    |   movel(p[0.465893, -0.053931, -0.000100, 0.000000, -3.141593, 0.000000],accel_mss,speed_ms,0,0.000)
    |   movel(p[0.464835, -0.052791, -0.000100, 0.000000, -3.141593, 0.000000],accel_mss,speed_ms,0,0.001)
    |   movel(p[0.463851, -0.051647, -0.000100, 0.000000, -3.141593, 0.000000],accel_mss,speed_ms,0,0.001)
    |   movel(p[0.463361, -0.050896, -0.000100, 0.000000, -3.141593, 0.000000],accel_mss,speed_ms,0,0.000)
    |   movel(p[0.463213, -0.050560, -0.000100, 0.000000, -3.141593, 0.000000],accel_mss,speed_ms,0,0.000)
    |   movel(p[0.463098, -0.050199, -0.000100, 0.000000, -3.141593, 0.000000],accel_mss,speed_ms,0,0.000)
    |   movel(p[0.463025, -0.049844, -0.000100, 0.000000, -3.141593, 0.000000],accel_mss,speed_ms,0,0.000)
    |   movel(p[0.463001, -0.049520, -0.000100, 0.000000, -3.141593, 0.000000],accel_mss,speed_ms,0,0.000)
    |   movel(p[0.462988, -0.049209, -0.000100, 0.000000, -3.141593, 0.000000],accel_mss,speed_ms,0,0.000)
    |   movel(p[0.462948, -0.048819, -0.000100, 0.000000, -3.141593, 0.000000],accel_mss,speed_ms,0,0.000)
    |   movel(p[0.462890, -0.048420, -0.000100, 0.000000, 3.141593, 0.000000],accel_mss,speed_ms,0,0.000)
    |   movel(p[0.462821, -0.048073, -0.000100, 0.000000, 3.141593, 0.000000],accel_mss,speed_ms,0,0.000)
    |   movel(p[0.462724, -0.047613, -0.000100, 0.000000, -3.141593, 0.000000],accel_mss,speed_ms,0,0.000)
    |   movel(p[0.462714, -0.047386, -0.000100, 0.000000, 3.141593, 0.000000],accel_mss,speed_ms,0,0.000)
    |   movel(p[0.462774, -0.047234, -0.000100, 0.000000, -3.141593, 0.000000],accel_mss,speed_ms,0,0.000)
    |   movel(p[0.462918, -0.047091, -0.000100, 0.000000, -3.141593, 0.000000],accel_mss,speed_ms,0,0.000)
    |   movel(p[0.463032, -0.047019, -0.000100, 0.000000, -3.141593, 0.000000],accel_mss,speed_ms,0,0.000)
    |   movel(p[0.463146, -0.046968, -0.000100, 0.000000, -3.141593, 0.000000],accel_mss,speed_ms,0,0.000)
    |   movel(p[0.463245, -0.046945, -0.000100, 0.000000, -3.141593, 0.000000],accel_mss,speed_ms,0,0.000)
    |   movel(p[0.463376, -0.046956, -0.000100, 0.000000, -3.141593, 0.000000],accel_mss,speed_ms,0,0.000)
    |   movel(p[0.463547, -0.046827, -0.000100, 0.000000, -3.141593, 0.000000],accel_mss,speed_ms,0,0.000)
    |   movel(p[0.463749, -0.046646, -0.000100, 0.000000, -3.141593, 0.000000],accel_mss,speed_ms,0,0.000)
    |   movel(p[0.463969, -0.046417, -0.000100, 0.000000, -3.141593, 0.000000],accel_mss,speed_ms,0,0.000)
    |   movel(p[0.464381, -0.046019, -0.000100, 0.000000, -3.141593, 0.000000],accel_mss,speed_ms,0,0.000)
    |   movel(p[0.464651, -0.045948, -0.000100, 0.000000, 3.141593, 0.000000],accel_mss,speed_ms,0,0.000)
    |   movel(p[0.464889, -0.046112, -0.000100, 0.000000, -3.141593, 0.000000],accel_mss,speed_ms,0,0.000)
    |   movel(p[0.465184, -0.046650, -0.000100, 0.000000, -3.141593, 0.000000],accel_mss,speed_ms,0,0.000)
    |   movel(p[0.465308, -0.047062, -0.000100, 0.000000, 3.141593, 0.000000],accel_mss,speed_ms,0,0.000)
    |   movel(p[0.465283, -0.047444, -0.000100, 0.000000, 3.141593, 0.000000],accel_mss,speed_ms,0,0.000)
    |   movel(p[0.465098, -0.047820, -0.000100, 0.000000, -3.141593, 0.000000],accel_mss,speed_ms,0,0.000)
    |   movel(p[0.464742, -0.048218, -0.000100, 0.000000, -3.141593, 0.000000],accel_mss,speed_ms,0,0.000)
    |   movel(p[0.464491, -0.048534, -0.000100, 0.000000, -3.141593, 0.000000],accel_mss,speed_ms,0,0.000)
    |   movel(p[0.464362, -0.048895, -0.000100, 0.000000, -3.141593, 0.000000],accel_mss,speed_ms,0,0.000)
    |   movel(p[0.464394, -0.049167, -0.000100, 0.000000, -3.141593, 0.000000],accel_mss,speed_ms,0,0.000)
    |   movel(p[0.464563, -0.049279, -0.000100, 0.000000, -3.141593, 0.000000],accel_mss,speed_ms,0,0.000)
    |   movel(p[0.464679, -0.049242, -0.000100, 0.000000, -3.141593, 0.000000],accel_mss,speed_ms,0,0.000)
    |   movel(p[0.464892, -0.049075, -0.000100, 0.000000, 3.141593, 0.000000],accel_mss,speed_ms,0,0.000)
    |   movel(p[0.465136, -0.048852, -0.000100, 0.000000, -3.141593, 0.000000],accel_mss,speed_ms,0,0.000)
    |   movel(p[0.465385, -0.048586, -0.000100, 0.000000, 3.141593, 0.000000],accel_mss,speed_ms,0,0.000)
    |   movel(p[0.465794, -0.048130, -0.000100, 0.000000, -3.141593, 0.000000],accel_mss,speed_ms,0,0.000)
    |   movel(p[0.465936, -0.048028, -0.000100, 0.000000, 3.141593, 0.000000],accel_mss,speed_ms,0,0.000)
    |   movel(p[0.466037, -0.048055, -0.000100, 0.000000, -3.141593, 0.000000],accel_mss,speed_ms,0,0.000)
    |   movel(p[0.466147, -0.048249, -0.000100, 0.000000, 3.141593, 0.000000],accel_mss,speed_ms,0,0.000)
    |   movel(p[0.466218, -0.048402, -0.000100, 0.000000, -3.141593, 0.000000],accel_mss,speed_ms,0,0.000)
    |   movel(p[0.466305, -0.048569, -0.000100, 0.000000, -3.141593, 0.000000],accel_mss,speed_ms,0,0.000)
    |   movel(p[0.466394, -0.048724, -0.000100, 0.000000, -3.141593, 0.000000],accel_mss,speed_ms,0,0.000)
    |   movel(p[0.466470, -0.048840, -0.000100, 0.000000, -3.141593, 0.000000],accel_mss,speed_ms,0,0.000)
    |   movel(p[0.466537, -0.048985, -0.000100, 0.000000, -3.141593, 0.000000],accel_mss,speed_ms,0,0.000)
    |   movel(p[0.466547, -0.049150, -0.000100, 0.000000, -3.141593, 0.000000],accel_mss,speed_ms,0,0.000)
    |   movel(p[0.466496, -0.049362, -0.000100, 0.000000, -3.141593, 0.000000],accel_mss,speed_ms,0,0.000)
    |   movel(p[0.466370, -0.049665, -0.000100, 0.000000, -3.141593, 0.000000],accel_mss,speed_ms,0,0.000)
    |   movel(p[0.466251, -0.049909, -0.000100, 0.000000, 3.141593, 0.000000],accel_mss,speed_ms,0,0.000)
    |   movel(p[0.466117, -0.050154, -0.000100, 0.000000, -3.141593, 0.000000],accel_mss,speed_ms,0,0.000)
    |   movel(p[0.465988, -0.050369, -0.000100, 0.000000, -3.141593, 0.000000],accel_mss,speed_ms,0,0.000)
    |   movel(p[0.465888, -0.050504, -0.000100, 0.000000, -3.141593, 0.000000],accel_mss,speed_ms,0,0.000)
    |   movel(p[0.465811, -0.050625, -0.000100, 0.000000, -3.141593, 0.000000],accel_mss,speed_ms,0,0.000)
    |   movel(p[0.465753, -0.050783, -0.000100, 0.000000, -3.141593, 0.000000],accel_mss,speed_ms,0,0.000)
    |   movel(p[0.465723, -0.050952, -0.000100, 0.000000, -3.141593, 0.000000],accel_mss,speed_ms,0,0.000)
    |   movel(p[0.465726, -0.051104, -0.000100, 0.000000, -3.141593, 0.000000],accel_mss,speed_ms,0,0.000)
    |   movel(p[0.465772, -0.051280, -0.000100, 0.000000, -3.141593, 0.000000],accel_mss,speed_ms,0,0.000)
    |   movel(p[0.465851, -0.051379, -0.000100, 0.000000, -3.141593, 0.000000],accel_mss,speed_ms,0,0.000)
    |   movel(p[0.465984, -0.051424, -0.000100, 0.000000, -3.141593, 0.000000],accel_mss,speed_ms,0,0.000)
    |   movel(p[0.466209, -0.051423, -0.000100, 0.000000, -3.141593, 0.000000],accel_mss,speed_ms,0,0.000)
    |   movel(p[0.466401, -0.051387, -0.000100, 0.000000, -3.141593, 0.000000],accel_mss,speed_ms,0,0.000)
    |   movel(p[0.466618, -0.051304, -0.000100, 0.000000, 3.141593, 0.000000],accel_mss,speed_ms,0,0.000)
    |   movel(p[0.466827, -0.051191, -0.000100, 0.000000, 3.141593, 0.000000],accel_mss,speed_ms,0,0.000)
    |   movel(p[0.466992, -0.051063, -0.000100, 0.000000, -3.141593, 0.000000],accel_mss,speed_ms,0,0.000)
    |   movel(p[0.467187, -0.050897, -0.000100, 0.000000, 3.141593, 0.000000],accel_mss,speed_ms,0,0.000)
    |   movel(p[0.467319, -0.050833, -0.000100, 0.000000, -3.141593, 0.000000],accel_mss,speed_ms,0,0.000)
    |   movel(p[0.467437, -0.050843, -0.000100, 0.000000, -3.141593, 0.000000],accel_mss,speed_ms,0,0.000)
    |   movel(p[0.467571, -0.050925, -0.000100, 0.000000, -3.141593, 0.000000],accel_mss,speed_ms,0,0.000)
    |   movel(p[0.467659, -0.051011, -0.000100, 0.000000, -3.141593, 0.000000],accel_mss,speed_ms,0,0.000)
    |   movel(p[0.467733, -0.051113, -0.000100, 0.000000, -3.141593, 0.000000],accel_mss,speed_ms,0,0.000)
    |   movel(p[0.467784, -0.051213, -0.000100, 0.000000, 3.141593, 0.000000],accel_mss,speed_ms,0,0.000)
    |   movel(p[0.468014, -0.051722, -0.000100, 0.000000, -3.141593, 0.000000],accel_mss,speed_ms,0,0.000)
    |   movel(p[0.468764, -0.052182, -0.000100, 0.000000, -3.141593, 0.000000],accel_mss,speed_ms,0,0.000)
    |   movel(p[0.469662, -0.052521, -0.000100, 0.000000, 3.141593, 0.000000],accel_mss,speed_ms,0,0.000)
    |   movel(p[0.470426, -0.052584, -0.000100, 0.000000, -3.141593, 0.000000],accel_mss,speed_ms,0,0.000)
    |   movel(p[0.470557, -0.052560, -0.000100, 0.000000, 3.141593, 0.000000],accel_mss,speed_ms,0,0.000)
    |   movel(p[0.470502, -0.052461, -0.000100, 0.000000, -3.141593, 0.000000],accel_mss,speed_ms,0,0.000)
    |   movel(p[0.470257, -0.052349, -0.000100, 0.000000, 3.141593, 0.000000],accel_mss,speed_ms,0,0.000)
    |   movel(p[0.470044, -0.052237, -0.000100, 0.000000, -3.141593, 0.000000],accel_mss,speed_ms,0,0.000)
    |   movel(p[0.469789, -0.052067, -0.000100, 0.000000, -3.141593, 0.000000],accel_mss,speed_ms,0,0.000)
    |   movel(p[0.469535, -0.051871, -0.000100, 0.000000, -3.141593, 0.000000],accel_mss,speed_ms,0,0.000)
    |   movel(p[0.469322, -0.051678, -0.000100, 0.000000, -3.141593, 0.000000],accel_mss,speed_ms,0,0.000)
    |   movel(p[0.469017, -0.051335, -0.000100, 0.000000, -3.141593, 0.000000],accel_mss,speed_ms,0,0.000)
    |   movel(p[0.468787, -0.050993, -0.000100, 0.000000, -3.141593, 0.000000],accel_mss,speed_ms,0,0.000)
    |   movel(p[0.468535, -0.050495, -0.000100, 0.000000, -3.141593, 0.000000],accel_mss,speed_ms,0,0.000)
    |   movel(p[0.468097, -0.049504, -0.000100, 0.000000, -3.141593, 0.000000],accel_mss,speed_ms,0,0.000)
    |   movel(p[0.467644, -0.048482, -0.000100, 0.000000, -3.141593, 0.000000],accel_mss,speed_ms,0,0.000)
    |   movel(p[0.467263, -0.047682, -0.000100, 0.000000, -3.141593, 0.000000],accel_mss,speed_ms,0,0.000)
    |   movel(p[0.466940, -0.047069, -0.000100, 0.000000, -3.141593, 0.000000],accel_mss,speed_ms,0,0.000)
    |   movel(p[0.466677, -0.046654, -0.000100, 0.000000, -3.141593, 0.000000],accel_mss,speed_ms,0,0.000)
    |   movel(p[0.466546, -0.046465, -0.000100, 0.000000, -3.141593, 0.000000],accel_mss,speed_ms,0,0.000)
    |   movel(p[0.466418, -0.046270, -0.000100, 0.000000, -3.141593, 0.000000],accel_mss,speed_ms,0,0.000)
    |   movel(p[0.466311, -0.046095, -0.000100, 0.000000, -3.141593, 0.000000],accel_mss,speed_ms,0,0.000)
    |   movel(p[0.466250, -0.045979, -0.000100, 0.000000, 3.141593, 0.000000],accel_mss,speed_ms,0,0.000)
    |   movel(p[0.466191, -0.045863, -0.000100, 0.000000, -3.141593, 0.000000],accel_mss,speed_ms,0,0.000)
    |   movel(p[0.466091, -0.045688, -0.000100, 0.000000, -3.141593, 0.000000],accel_mss,speed_ms,0,0.000)
    |   movel(p[0.465972, -0.045493, -0.000100, 0.000000, -3.141593, 0.000000],accel_mss,speed_ms,0,0.000)
    |   movel(p[0.465851, -0.045304, -0.000100, 0.000000, -3.141593, 0.000000],accel_mss,speed_ms,0,0.000)
    |   movel(p[0.465728, -0.045110, -0.000100, 0.000000, -3.141593, 0.000000],accel_mss,speed_ms,0,0.000)
    |   movel(p[0.465602, -0.044898, -0.000100, 0.000000, 3.141593, 0.000000],accel_mss,speed_ms,0,0.000)
    |   movel(p[0.465492, -0.044700, -0.000100, 0.000000, -3.141593, 0.000000],accel_mss,speed_ms,0,0.000)
    |   movel(p[0.465420, -0.044554, -0.000100, 0.000000, -3.141593, 0.000000],accel_mss,speed_ms,0,0.000)
    |   movel(p[0.465263, -0.044299, -0.000100, 0.000000, -3.141593, 0.000000],accel_mss,speed_ms,0,0.000)
    |   movel(p[0.465028, -0.044054, -0.000100, 0.000000, -3.141593, 0.000000],accel_mss,speed_ms,0,0.000)
    |   movel(p[0.464698, -0.043807, -0.000100, 0.000000, -3.141593, 0.000000],accel_mss,speed_ms,0,0.000)
    |   movel(p[0.464252, -0.043540, -0.000100, 0.000000, -3.141593, 0.000000],accel_mss,speed_ms,0,0.000)
    |   movel(p[0.463697, -0.043350, -0.000100, 0.000000, -3.141593, 0.000000],accel_mss,speed_ms,0,0.000)
    |   movel(p[0.462896, -0.043284, -0.000100, 0.000000, -3.141593, 0.000000],accel_mss,speed_ms,0,0.000)
    |   movel(p[0.461992, -0.043334, -0.000100, 0.000000, -3.141593, 0.000000],accel_mss,speed_ms,0,0.000)
    |   movel(p[0.461101, -0.043504, -0.000100, 0.000000, -3.141593, 0.000000],accel_mss,speed_ms,0,0.000)
    |   movel(p[0.460265, -0.043707, -0.000100, 0.000000, -3.141593, 0.000000],accel_mss,speed_ms,0,0.000)
    |   movel(p[0.460020, -0.043670, -0.000100, 0.000000, 3.141593, 0.000000],accel_mss,speed_ms,0,0.000)
    |   movel(p[0.459904, -0.043483, -0.000100, 0.000000, -3.141593, 0.000000],accel_mss,speed_ms,0,0.000)
    |   movel(p[0.459894, -0.042823, -0.000100, 0.000000, -3.141593, 0.000000],accel_mss,speed_ms,0,0.000)
    |   movel(p[0.459902, -0.042370, -0.000100, 0.000000, -3.141593, 0.000000],accel_mss,speed_ms,0,0.000)
    |   movel(p[0.459911, -0.041917, -0.000100, 0.000000, -3.141593, 0.000000],accel_mss,speed_ms,0,0.000)
    |   movel(p[0.459479, -0.041489, -0.000100, 0.000000, 3.141593, 0.000000],accel_mss,speed_ms,0,0.000)
    |   movel(p[0.459048, -0.041061, -0.000100, 0.000000, -3.141593, 0.000000],accel_mss,speed_ms,0,0.000)
    |   movel(p[0.458516, -0.040544, -0.000100, 0.000000, -3.141593, 0.000000],accel_mss,speed_ms,0,0.000)
    |   movel(p[0.458286, -0.040375, -0.000100, 0.000000, -3.141593, 0.000000],accel_mss,speed_ms,0,0.000)
    |   movel(p[0.458130, -0.040364, -0.000100, 0.000000, -3.141593, 0.000000],accel_mss,speed_ms,0,0.000)
    |   movel(p[0.457983, -0.040475, -0.000100, 0.000000, -3.141593, 0.000000],accel_mss,speed_ms,0,0.000)
    |   movel(p[0.457901, -0.040642, -0.000100, 0.000000, 3.141593, 0.000000],accel_mss,speed_ms,0,0.000)
    |   movel(p[0.457835, -0.040932, -0.000100, 0.000000, -3.141593, 0.000000],accel_mss,speed_ms,0,0.000)
    |   movel(p[0.457791, -0.041287, -0.000100, 0.000000, -3.141593, 0.000000],accel_mss,speed_ms,0,0.000)
    |   movel(p[0.457774, -0.041675, -0.000100, 0.000000, -3.141593, 0.000000],accel_mss,speed_ms,0,0.000)
    |   movel(p[0.457772, -0.042046, -0.000100, 0.000000, -3.141593, 0.000000],accel_mss,speed_ms,0,0.000)
    |   movel(p[0.457768, -0.042392, -0.000100, 0.000000, -3.141593, 0.000000],accel_mss,speed_ms,0,0.000)
    |   movel(p[0.457764, -0.042683, -0.000100, 0.000000, -3.141593, 0.000000],accel_mss,speed_ms,0,0.000)
    |   movel(p[0.457760, -0.042812, -0.000100, 0.000000, -3.141593, 0.000000],accel_mss,speed_ms,0,0.000)
    |   movel(p[0.457706, -0.042908, -0.000100, 0.000000, -3.141593, 0.000000],accel_mss,speed_ms,0,0.000)
    |   movel(p[0.457569, -0.042961, -0.000100, 0.000000, -3.141593, 0.000000],accel_mss,speed_ms,0,0.000)
    |   movel(p[0.457315, -0.042972, -0.000100, 0.000000, -3.141593, 0.000000],accel_mss,speed_ms,0,0.000)
    |   movel(p[0.456863, -0.042940, -0.000100, 0.000000, -3.141593, 0.000000],accel_mss,speed_ms,0,0.000)
    |   movel(p[0.456466, -0.042918, -0.000100, 0.000000, -3.141593, 0.000000],accel_mss,speed_ms,0,0.000)
    |   movel(p[0.456116, -0.042929, -0.000100, 0.000000, -3.141593, 0.000000],accel_mss,speed_ms,0,0.000)
    |   movel(p[0.455826, -0.042970, -0.000100, 0.000000, -3.141593, 0.000000],accel_mss,speed_ms,0,0.000)
    |   movel(p[0.455621, -0.043043, -0.000100, 0.000000, -3.141593, 0.000000],accel_mss,speed_ms,0,0.000)
    |   movel(p[0.455348, -0.043146, -0.000100, 0.000000, -3.141593, 0.000000],accel_mss,speed_ms,0,0.000)
    |   movel(p[0.455101, -0.043158, -0.000100, 0.000000, -3.141593, 0.000000],accel_mss,speed_ms,0,0.000)
    |   movel(p[0.454859, -0.043077, -0.000100, 0.000000, -3.141593, 0.000000],accel_mss,speed_ms,0,0.000)
    |   movel(p[0.454601, -0.042898, -0.000100, 0.000000, -3.141593, 0.000000],accel_mss,speed_ms,0,0.000)
    |   movel(p[0.454453, -0.042792, -0.000100, 0.000000, -3.141593, 0.000000],accel_mss,speed_ms,0,0.000)
    |   movel(p[0.454095, -0.042581, -0.000100, 0.000000, -3.141593, 0.000000],accel_mss,speed_ms,0,0.000)
    |   movel(p[0.453664, -0.042338, -0.000100, 0.000000, -3.141593, 0.000000],accel_mss,speed_ms,0,0.000)
    |   movel(p[0.453196, -0.042087, -0.000100, 0.000000, -3.141593, 0.000000],accel_mss,speed_ms,0,0.000)
    |   movel(p[0.451387, -0.041339, -0.000100, 0.000000, -3.141593, 0.000000],accel_mss,speed_ms,0,0.001)
    |   movel(p[0.449147, -0.040777, -0.000100, 0.000000, -3.141593, 0.000000],accel_mss,speed_ms,0,0.001)
    |   movel(p[0.446912, -0.040477, -0.000100, 0.000000, 3.141593, 0.000000],accel_mss,speed_ms,0,0.001)
    |   movel(p[0.445133, -0.040539, -0.000100, 0.000000, -3.141593, 0.000000],accel_mss,speed_ms,0,0.001)
    |   movel(p[0.443736, -0.040810, -0.000100, 0.000000, -3.141593, 0.000000],accel_mss,speed_ms,0,0.001)
    |   movel(p[0.442479, -0.041187, -0.000100, 0.000000, -3.141593, 0.000000],accel_mss,speed_ms,0,0.001)
    |   movel(p[0.441469, -0.041626, -0.000100, 0.000000, -3.141593, 0.000000],accel_mss,speed_ms,0,0.000)
    |   movel(p[0.440872, -0.042084, -0.000100, 0.000000, 3.141593, 0.000000],accel_mss,speed_ms,0,0.000)
    |   movel(p[0.440734, -0.042220, -0.000100, 0.000000, 3.141593, 0.000000],accel_mss,speed_ms,0,0.000)
    |   movel(p[0.440563, -0.042355, -0.000100, 0.000000, -3.141593, 0.000000],accel_mss,speed_ms,0,0.000)
    |   movel(p[0.440387, -0.042470, -0.000100, 0.000000, -3.141593, 0.000000],accel_mss,speed_ms,0,0.000)
    |   movel(p[0.440235, -0.042543, -0.000100, 0.000000, -3.141593, 0.000000],accel_mss,speed_ms,0,0.000)
    |   movel(p[0.440096, -0.042618, -0.000100, 0.000000, -3.141593, 0.000000],accel_mss,speed_ms,0,0.000)
    |   movel(p[0.439957, -0.042735, -0.000100, 0.000000, 3.141593, 0.000000],accel_mss,speed_ms,0,0.000)
    |   movel(p[0.439840, -0.042874, -0.000100, 0.000000, -3.141593, 0.000000],accel_mss,speed_ms,0,0.000)
    |   movel(p[0.439765, -0.043014, -0.000100, 0.000000, -3.141593, 0.000000],accel_mss,speed_ms,0,0.000)
    |   movel(p[0.439692, -0.043165, -0.000100, 0.000000, 3.141593, 0.000000],accel_mss,speed_ms,0,0.000)
    |   movel(p[0.439577, -0.043341, -0.000100, 0.000000, -3.141593, 0.000000],accel_mss,speed_ms,0,0.000)
    |   movel(p[0.439442, -0.043512, -0.000100, 0.000000, -3.141593, 0.000000],accel_mss,speed_ms,0,0.000)
    |   movel(p[0.439306, -0.043650, -0.000100, 0.000000, -3.141593, 0.000000],accel_mss,speed_ms,0,0.000)
    |   movel(p[0.439069, -0.043925, -0.000100, 0.000000, -3.141593, 0.000000],accel_mss,speed_ms,0,0.000)
    |   movel(p[0.438803, -0.044367, -0.000100, 0.000000, -3.141593, 0.000000],accel_mss,speed_ms,0,0.000)
    |   movel(p[0.438526, -0.044932, -0.000100, 0.000000, 3.141593, 0.000000],accel_mss,speed_ms,0,0.000)
    |   movel(p[0.438251, -0.045603, -0.000100, 0.000000, -3.141593, 0.000000],accel_mss,speed_ms,0,0.000)
    |   movel(p[0.438049, -0.045882, -0.000100, 0.000000, -3.141593, 0.000000],accel_mss,speed_ms,0,0.000)
    |   movel(p[0.437776, -0.045945, -0.000100, 0.000000, -3.141593, 0.000000],accel_mss,speed_ms,0,0.000)
    |   movel(p[0.437406, -0.045762, -0.000100, 0.000000, -3.141593, 0.000000],accel_mss,speed_ms,0,0.000)
    |   movel(p[0.436894, -0.045290, -0.000100, 0.000000, -3.141593, 0.000000],accel_mss,speed_ms,0,0.000)
    |   movel(p[0.436616, -0.045016, -0.000100, 0.000000, -3.141593, 0.000000],accel_mss,speed_ms,0,0.000)
    |   movel(p[0.436334, -0.044763, -0.000100, 0.000000, -3.141593, 0.000000],accel_mss,speed_ms,0,0.000)
    |   movel(p[0.436082, -0.044558, -0.000100, 0.000000, 3.141593, 0.000000],accel_mss,speed_ms,0,0.000)
    |   movel(p[0.435926, -0.044463, -0.000100, 0.000000, -3.141593, 0.000000],accel_mss,speed_ms,0,0.000)
    |   movel(p[0.435779, -0.044389, -0.000100, 0.000000, -3.141593, 0.000000],accel_mss,speed_ms,0,0.000)
    |   movel(p[0.435582, -0.044278, -0.000100, 0.000000, -3.141593, 0.000000],accel_mss,speed_ms,0,0.000)
    |   movel(p[0.435370, -0.044152, -0.000100, 0.000000, -3.141593, 0.000000],accel_mss,speed_ms,0,0.000)
    |   movel(p[0.435176, -0.044028, -0.000100, 0.000000, -3.141593, 0.000000],accel_mss,speed_ms,0,0.000)
    |   movel(p[0.434461, -0.043604, -0.000100, 0.000000, 3.141593, 0.000000],accel_mss,speed_ms,0,0.000)
    |   movel(p[0.433429, -0.043079, -0.000100, 0.000000, 3.141593, 0.000000],accel_mss,speed_ms,0,0.000)
    |   movel(p[0.432404, -0.042596, -0.000100, 0.000000, 3.141593, 0.000000],accel_mss,speed_ms,0,0.000)
    |   movel(p[0.431959, -0.042462, -0.000100, 0.000000, -3.141593, 0.000000],accel_mss,speed_ms,0,0.000)
    |   movel(p[0.430393, -0.042224, -0.000100, 0.000000, -3.141593, 0.000000],accel_mss,speed_ms,0,0.001)
    |   movel(p[0.429462, -0.042122, -0.000100, 0.000000, -3.141593, 0.000000],accel_mss,speed_ms,0,0.000)
    |   movel(p[0.428675, -0.042100, -0.000100, 0.000000, -3.141593, 0.000000],accel_mss,speed_ms,0,0.000)
    |   movel(p[0.427707, -0.042143, -0.000100, 0.000000, 3.141593, 0.000000],accel_mss,speed_ms,0,0.000)
    |   movel(p[0.427099, -0.042188, -0.000100, 0.000000, -3.141593, 0.000000],accel_mss,speed_ms,0,0.000)
    |   movel(p[0.426537, -0.042231, -0.000100, 0.000000, -3.141593, 0.000000],accel_mss,speed_ms,0,0.000)
    |   movel(p[0.426067, -0.042270, -0.000100, 0.000000, -3.141593, 0.000000],accel_mss,speed_ms,0,0.000)
    |   movel(p[0.425876, -0.042291, -0.000100, 0.000000, -3.141593, 0.000000],accel_mss,speed_ms,0,0.000)
    |   movel(p[0.424163, -0.042642, -0.000100, 0.000000, -3.141593, 0.000000],accel_mss,speed_ms,0,0.001)
    |   movel(p[0.422697, -0.043203, -0.000100, 0.000000, -3.141593, 0.000000],accel_mss,speed_ms,0,0.001)
    |   movel(p[0.421369, -0.044026, -0.000100, 0.000000, -3.141593, 0.000000],accel_mss,speed_ms,0,0.001)
    |   movel(p[0.420072, -0.045167, -0.000100, 0.000000, -3.141593, 0.000000],accel_mss,speed_ms,0,0.001)
    |   movel(p[0.419586, -0.045650, -0.000100, 0.000000, 3.141593, 0.000000],accel_mss,speed_ms,0,0.000)
    |   movel(p[0.419159, -0.046058, -0.000100, 0.000000, -3.141593, 0.000000],accel_mss,speed_ms,0,0.000)
    |   movel(p[0.418787, -0.046400, -0.000100, 0.000000, -3.141593, 0.000000],accel_mss,speed_ms,0,0.000)
    |   movel(p[0.418627, -0.046370, -0.000100, 0.000000, -3.141593, 0.000000],accel_mss,speed_ms,0,0.000)
    |   movel(p[0.418632, -0.046249, -0.000100, 0.000000, -3.141593, 0.000000],accel_mss,speed_ms,0,0.000)
    |   movel(p[0.418775, -0.046039, -0.000100, 0.000000, -3.141593, 0.000000],accel_mss,speed_ms,0,0.000)
    |   movel(p[0.419051, -0.045754, -0.000100, 0.000000, -3.141593, 0.000000],accel_mss,speed_ms,0,0.000)
    |   movel(p[0.419223, -0.045578, -0.000100, 0.000000, -3.141593, 0.000000],accel_mss,speed_ms,0,0.000)
    |   movel(p[0.419368, -0.045406, -0.000100, 0.000000, -3.141593, 0.000000],accel_mss,speed_ms,0,0.000)
    |   movel(p[0.419476, -0.045257, -0.000100, 0.000000, -3.141593, 0.000000],accel_mss,speed_ms,0,0.000)
    |   movel(p[0.419626, -0.044852, -0.000100, 0.000000, -3.141593, 0.000000],accel_mss,speed_ms,0,0.000)
    |   movel(p[0.421392, -0.042927, -0.000100, 0.000000, -3.141593, 0.000000],accel_mss,speed_ms,0,blend_radius_m)
    |   movel(p[0.423178, -0.041005, -0.000100, 0.000000, -3.141593, 0.000000],accel_mss,speed_ms,0,blend_radius_m)
    |   movel(p[0.423470, -0.040879, -0.000100, 0.000000, -3.141593, 0.000000],accel_mss,speed_ms,0,0.000)
    |   movel(p[0.423568, -0.040846, -0.000100, 0.000000, -3.141593, 0.000000],accel_mss,speed_ms,0,0.000)
    |   movel(p[0.423805, -0.040659, -0.000100, 0.000000, -3.141593, 0.000000],accel_mss,speed_ms,0,0.000)
    |   movel(p[0.424080, -0.040416, -0.000100, 0.000000, 3.141593, 0.000000],accel_mss,speed_ms,0,0.000)
    |   movel(p[0.424376, -0.040129, -0.000100, 0.000000, -3.141593, 0.000000],accel_mss,speed_ms,0,0.000)
    |   movel(p[0.424668, -0.039842, -0.000100, 0.000000, -3.141593, 0.000000],accel_mss,speed_ms,0,0.000)
    |   movel(p[0.424937, -0.039599, -0.000100, 0.000000, 3.141593, 0.000000],accel_mss,speed_ms,0,0.000)
    |   movel(p[0.425167, -0.039408, -0.000100, 0.000000, -3.141593, 0.000000],accel_mss,speed_ms,0,0.000)
    |   movel(p[0.425335, -0.039352, -0.000100, 0.000000, -3.141593, 0.000000],accel_mss,speed_ms,0,0.000)
    |   movel(p[0.425593, -0.039167, -0.000100, 0.000000, 3.141593, 0.000000],accel_mss,speed_ms,0,0.000)
    |   movel(p[0.425897, -0.038933, -0.000100, 0.000000, -3.141593, 0.000000],accel_mss,speed_ms,0,0.000)
    |   movel(p[0.426230, -0.038657, -0.000100, 0.000000, -3.141593, 0.000000],accel_mss,speed_ms,0,0.000)
    |   movel(p[0.426595, -0.038361, -0.000100, 0.000000, -3.141593, 0.000000],accel_mss,speed_ms,0,0.000)
    |   movel(p[0.426991, -0.038071, -0.000100, 0.000000, 3.141593, 0.000000],accel_mss,speed_ms,0,0.000)
    |   movel(p[0.427361, -0.037825, -0.000100, 0.000000, -3.141593, 0.000000],accel_mss,speed_ms,0,0.000)
    |   movel(p[0.427632, -0.037678, -0.000100, 0.000000, -3.141593, 0.000000],accel_mss,speed_ms,0,0.000)
    |   movel(p[0.427851, -0.037569, -0.000100, 0.000000, -3.141593, 0.000000],accel_mss,speed_ms,0,0.000)
    |   movel(p[0.428049, -0.037456, -0.000100, 0.000000, -3.141593, 0.000000],accel_mss,speed_ms,0,0.000)
    |   movel(p[0.428208, -0.037352, -0.000100, 0.000000, 3.141593, 0.000000],accel_mss,speed_ms,0,0.000)
    |   movel(p[0.428330, -0.037218, -0.000100, 0.000000, -3.141593, 0.000000],accel_mss,speed_ms,0,0.000)
    |   movel(p[0.428452, -0.037125, -0.000100, 0.000000, -3.141593, 0.000000],accel_mss,speed_ms,0,0.000)
    |   movel(p[0.428603, -0.037026, -0.000100, 0.000000, -3.141593, 0.000000],accel_mss,speed_ms,0,0.000)
    |   movel(p[0.428766, -0.036934, -0.000100, 0.000000, -3.141593, 0.000000],accel_mss,speed_ms,0,0.000)
    |   movel(p[0.429000, -0.036811, -0.000100, 0.000000, 3.141593, 0.000000],accel_mss,speed_ms,0,0.000)
    |   movel(p[0.429430, -0.036585, -0.000100, 0.000000, -3.141593, 0.000000],accel_mss,speed_ms,0,0.000)
    |   movel(p[0.429933, -0.036321, -0.000100, 0.000000, -3.141593, 0.000000],accel_mss,speed_ms,0,0.000)
    |   movel(p[0.430451, -0.036048, -0.000100, 0.000000, -3.141593, 0.000000],accel_mss,speed_ms,0,0.000)
    |   movel(p[0.430984, -0.035777, -0.000100, 0.000000, -3.141593, 0.000000],accel_mss,speed_ms,0,0.000)
    |   movel(p[0.431528, -0.035517, -0.000100, 0.000000, -3.141593, 0.000000],accel_mss,speed_ms,0,0.000)
    |   movel(p[0.432013, -0.035301, -0.000100, 0.000000, -3.141593, 0.000000],accel_mss,speed_ms,0,0.000)
    |   movel(p[0.432326, -0.035183, -0.000100, 0.000000, 3.141593, 0.000000],accel_mss,speed_ms,0,0.000)
    |   movel(p[0.432567, -0.035101, -0.000100, 0.000000, -3.141593, 0.000000],accel_mss,speed_ms,0,0.000)
    |   movel(p[0.432794, -0.035014, -0.000100, 0.000000, -3.141593, 0.000000],accel_mss,speed_ms,0,0.000)
    |   movel(p[0.432983, -0.034933, -0.000100, 0.000000, -3.141593, 0.000000],accel_mss,speed_ms,0,0.000)
    |   movel(p[0.433076, -0.034879, -0.000100, 0.000000, -3.141593, 0.000000],accel_mss,speed_ms,0,0.000)
    |   movel(p[0.433419, -0.034699, -0.000100, 0.000000, -3.141593, 0.000000],accel_mss,speed_ms,0,0.000)
    |   movel(p[0.434424, -0.034366, -0.000100, 0.000000, -3.141593, 0.000000],accel_mss,speed_ms,0,0.000)
    |   movel(p[0.435617, -0.034006, -0.000100, 0.000000, -3.141593, 0.000000],accel_mss,speed_ms,0,0.000)
    |   movel(p[0.436901, -0.033659, -0.000100, 0.000000, -3.141593, 0.000000],accel_mss,speed_ms,0,0.001)
    |   movel(p[0.440327, -0.033025, -0.000100, 0.000000, -3.141593, 0.000000],accel_mss,speed_ms,0,blend_radius_m)
    |   movel(p[0.444164, -0.032779, -0.000100, 0.000000, -3.141593, 0.000000],accel_mss,speed_ms,0,blend_radius_m)
    |   movel(p[0.448043, -0.032923, -0.000100, 0.000000, -3.141593, 0.000000],accel_mss,speed_ms,0,blend_radius_m)
    |   movel(p[0.451601, -0.033464, -0.000100, 0.000000, 3.141593, 0.000000],accel_mss,speed_ms,0,blend_radius_m)
    |   movel(p[0.453044, -0.033799, -0.000100, 0.000000, -3.141593, 0.000000],accel_mss,speed_ms,0,0.001)
    |   movel(p[0.454520, -0.034184, -0.000100, 0.000000, -3.141593, 0.000000],accel_mss,speed_ms,0,0.001)
    |   movel(p[0.455867, -0.034563, -0.000100, 0.000000, -3.141593, 0.000000],accel_mss,speed_ms,0,0.001)
    |   movel(p[0.456172, -0.034719, -0.000100, 0.000000, -3.141593, 0.000000],accel_mss,speed_ms,0,0.000)
    |   movel(p[0.456267, -0.034777, -0.000100, 0.000000, -3.141593, 0.000000],accel_mss,speed_ms,0,0.000)
    |   movel(p[0.456457, -0.034860, -0.000100, 0.000000, -3.141593, 0.000000],accel_mss,speed_ms,0,0.000)
    |   movel(p[0.456685, -0.034949, -0.000100, 0.000000, 3.141593, 0.000000],accel_mss,speed_ms,0,0.000)
    |   movel(p[0.456926, -0.035030, -0.000100, 0.000000, -3.141593, 0.000000],accel_mss,speed_ms,0,0.000)
    |   movel(p[0.457819, -0.035379, -0.000100, 0.000000, -3.141593, 0.000000],accel_mss,speed_ms,0,0.000)
    |   movel(p[0.459590, -0.036225, -0.000100, 0.000000, -3.141593, 0.000000],accel_mss,speed_ms,0,0.001)
    |   movel(p[0.461358, -0.037107, -0.000100, 0.000000, -3.141593, 0.000000],accel_mss,speed_ms,0,0.001)
    |   movel(p[0.462040, -0.037531, -0.000100, 0.000000, -3.141593, 0.000000],accel_mss,speed_ms,0,0.000)
    |   movel(p[0.462229, -0.037664, -0.000100, 0.000000, -3.141593, 0.000000],accel_mss,speed_ms,0,0.000)
    |   movel(p[0.462412, -0.037777, -0.000100, 0.000000, -3.141593, 0.000000],accel_mss,speed_ms,0,0.000)
    |   movel(p[0.462570, -0.037860, -0.000100, 0.000000, -3.141593, 0.000000],accel_mss,speed_ms,0,0.000)
    |   movel(p[0.462729, -0.037898, -0.000100, 0.000000, -3.141593, 0.000000],accel_mss,speed_ms,0,0.000)
    |   movel(p[0.462840, -0.037967, -0.000100, 0.000000, 3.141593, 0.000000],accel_mss,speed_ms,0,0.000)
    |   movel(p[0.462961, -0.038064, -0.000100, 0.000000, -3.141593, 0.000000],accel_mss,speed_ms,0,0.000)
    |   movel(p[0.463076, -0.038179, -0.000100, 0.000000, -3.141593, 0.000000],accel_mss,speed_ms,0,0.000)
    |   movel(p[0.463192, -0.038294, -0.000100, 0.000000, -3.141593, 0.000000],accel_mss,speed_ms,0,0.000)
    |   movel(p[0.463319, -0.038391, -0.000100, 0.000000, -3.141593, 0.000000],accel_mss,speed_ms,0,0.000)
    |   movel(p[0.463437, -0.038459, -0.000100, 0.000000, -3.141593, 0.000000],accel_mss,speed_ms,0,0.000)
    |   movel(p[0.463613, -0.038502, -0.000100, 0.000000, -3.141593, 0.000000],accel_mss,speed_ms,0,0.000)
    |   movel(p[0.463750, -0.038589, -0.000100, 0.000000, -3.141593, 0.000000],accel_mss,speed_ms,0,0.000)
    |   movel(p[0.463903, -0.038710, -0.000100, 0.000000, -3.141593, 0.000000],accel_mss,speed_ms,0,0.000)
    |   movel(p[0.464051, -0.038854, -0.000100, 0.000000, -3.141593, 0.000000],accel_mss,speed_ms,0,0.000)
    |   movel(p[0.464201, -0.038997, -0.000100, 0.000000, 3.141593, 0.000000],accel_mss,speed_ms,0,0.000)
    |   movel(p[0.464361, -0.039119, -0.000100, 0.000000, -3.141593, 0.000000],accel_mss,speed_ms,0,0.000)
    |   movel(p[0.464508, -0.039204, -0.000100, 0.000000, -3.141593, 0.000000],accel_mss,speed_ms,0,0.000)
    |   movel(p[0.464611, -0.039229, -0.000100, 0.000000, -3.141593, 0.000000],accel_mss,speed_ms,0,0.000)
    |   movel(p[0.464940, -0.039364, -0.000100, 0.000000, 3.141593, 0.000000],accel_mss,speed_ms,0,0.000)
    |   movel(p[0.467208, -0.041623, -0.000100, 0.000000, -3.141593, 0.000000],accel_mss,speed_ms,0,blend_radius_m)
    |   movel(p[0.469465, -0.043893, -0.000100, 0.000000, -3.141593, 0.000000],accel_mss,speed_ms,0,blend_radius_m)
    |   movel(p[0.469601, -0.044221, -0.000100, 0.000000, 3.141593, 0.000000],accel_mss,speed_ms,0,0.000)
    |   movel(p[0.469621, -0.044321, -0.000100, 0.000000, -3.141593, 0.000000],accel_mss,speed_ms,0,0.000)
    |   movel(p[0.469686, -0.044448, -0.000100, 0.000000, -3.141593, 0.000000],accel_mss,speed_ms,0,0.000)
    |   movel(p[0.469781, -0.044580, -0.000100, 0.000000, -3.141593, 0.000000],accel_mss,speed_ms,0,0.000)
    |   movel(p[0.469892, -0.044696, -0.000100, 0.000000, -3.141593, 0.000000],accel_mss,speed_ms,0,0.000)
    |   movel(p[0.470011, -0.044829, -0.000100, 0.000000, -3.141593, 0.000000],accel_mss,speed_ms,0,0.000)
    |   movel(p[0.470126, -0.045010, -0.000100, 0.000000, -3.141593, 0.000000],accel_mss,speed_ms,0,0.000)
    |   movel(p[0.470221, -0.045208, -0.000100, 0.000000, -3.141593, 0.000000],accel_mss,speed_ms,0,0.000)
    |   movel(p[0.470279, -0.045393, -0.000100, 0.000000, -3.141593, 0.000000],accel_mss,speed_ms,0,0.000)
    |   movel(p[0.470326, -0.045565, -0.000100, 0.000000, -3.141593, 0.000000],accel_mss,speed_ms,0,0.000)
    |   movel(p[0.470389, -0.045725, -0.000100, 0.000000, -3.141593, 0.000000],accel_mss,speed_ms,0,0.000)
    |   movel(p[0.470458, -0.045853, -0.000100, 0.000000, 3.141593, 0.000000],accel_mss,speed_ms,0,0.000)
    |   movel(p[0.470779, -0.046211, -0.000100, 0.000000, -3.141593, 0.000000],accel_mss,speed_ms,0,0.000)
    |   movel(p[0.471394, -0.047619, -0.000100, 0.000000, -3.141593, 0.000000],accel_mss,speed_ms,0,0.001)
    |   movel(p[0.472003, -0.049141, -0.000100, 0.000000, -3.141593, 0.000000],accel_mss,speed_ms,0,0.001)
    |   movel(p[0.472489, -0.050554, -0.000100, 0.000000, -3.141593, 0.000000],accel_mss,speed_ms,0,0.001)
    |   movel(p[0.472833, -0.051729, -0.000100, 0.000000, -3.141593, 0.000000],accel_mss,speed_ms,0,0.000)
    |   movel(p[0.473221, -0.053215, -0.000100, 0.000000, -3.141593, 0.000000],accel_mss,speed_ms,0,0.001)
    |   movel(p[0.473563, -0.054635, -0.000100, 0.000000, -3.141593, 0.000000],accel_mss,speed_ms,0,0.001)
    |   movel(p[0.473710, -0.055429, -0.000100, 0.000000, -3.141593, 0.000000],accel_mss,speed_ms,0,0.000)
    |   movel(p[0.473745, -0.055714, -0.000100, 0.000000, -3.141593, 0.000000],accel_mss,speed_ms,0,0.000)
    |   movel(p[0.473792, -0.056185, -0.000100, 0.000000, -3.141593, 0.000000],accel_mss,speed_ms,0,0.000)
    |   movel(p[0.473842, -0.056725, -0.000100, 0.000000, -3.141593, 0.000000],accel_mss,speed_ms,0,0.000)
    |   movel(p[0.473887, -0.057266, -0.000100, 0.000000, -3.141593, 0.000000],accel_mss,speed_ms,0,0.000)
    |   movel(p[0.473940, -0.057923, -0.000100, 0.000000, -3.141593, 0.000000],accel_mss,speed_ms,0,0.000)
    |   movel(p[0.473992, -0.058579, -0.000100, 0.000000, -3.141593, 0.000000],accel_mss,speed_ms,0,0.000)
    |   movel(p[0.473616, -0.058579, -0.000100, 0.000000, 3.141593, 0.000000],accel_mss,speed_ms,0,0.000)
    |   movel(p[0.473241, -0.058579, -0.000100, 0.000000, 3.141593, 0.000000],accel_mss,speed_ms,0,0.000)
    |   movel(p[0.472392, -0.058631, -0.000100, 0.000000, 3.141593, 0.000000],accel_mss,speed_ms,0,0.000)
    |   movel(p[0.471238, -0.058802, -0.000100, 0.000000, -3.141593, 0.000000],accel_mss,speed_ms,0,0.000)
    |   movel(p[0.470098, -0.059028, -0.000100, 0.000000, -3.141593, 0.000000],accel_mss,speed_ms,0,0.000)
    |   movel(p[0.469296, -0.059262, -0.000100, 0.000000, -3.141593, 0.000000],accel_mss,speed_ms,0,0.000)
    |   movel(p[0.469027, -0.059357, -0.000100, 0.000000, -3.141593, 0.000000],accel_mss,speed_ms,0,0.000)
    |   movel(p[0.468772, -0.059443, -0.000100, 0.000000, -3.141593, 0.000000],accel_mss,speed_ms,0,0.000)
    |   movel(p[0.468556, -0.059511, -0.000100, 0.000000, -3.141593, 0.000000],accel_mss,speed_ms,0,0.000)
    |   movel(p[0.468453, -0.059536, -0.000100, 0.000000, -3.141593, 0.000000],accel_mss,speed_ms,0,0.000)
    |   movel(p[0.468272, -0.059608, -0.000100, 0.000000, -3.141593, 0.000000],accel_mss,speed_ms,0,0.000)
    |   movel(p[0.468168, -0.059669, -0.000100, 0.000000, -3.141593, 0.000000],accel_mss,speed_ms,0,0.000)
    |   movel(p[0.468077, -0.059736, -0.000100, 0.000000, -3.141593, 0.000000],accel_mss,speed_ms,0,0.000)
    |   movel(p[0.467973, -0.059808, -0.000100, 0.000000, -3.141593, 0.000000],accel_mss,speed_ms,0,0.000)
    |   movel(p[0.467822, -0.059883, -0.000100, 0.000000, -3.141593, 0.000000],accel_mss,speed_ms,0,0.000)
    |   movel(p[0.467654, -0.059951, -0.000100, 0.000000, -3.141593, 0.000000],accel_mss,speed_ms,0,0.000)
    |   movel(p[0.467493, -0.060000, -0.000100, 0.000000, -3.141593, 0.000000],accel_mss,speed_ms,0,0.000)
    |   movel(p[0.467019, -0.060219, -0.000100, 0.000000, -3.141593, 0.000000],accel_mss,speed_ms,0,0.000)
    |   movel(p[0.466394, -0.060719, -0.000100, 0.000000, -3.141593, 0.000000],accel_mss,speed_ms,0,0.000)
    |   movel(p[0.465818, -0.061299, -0.000100, 0.000000, -3.141593, 0.000000],accel_mss,speed_ms,0,0.000)
    |   movel(p[0.465488, -0.061799, -0.000100, 0.000000, -3.141593, 0.000000],accel_mss,speed_ms,0,0.000)
    |   movel(p[0.465276, -0.062191, -0.000100, 0.000000, 3.141593, 0.000000],accel_mss,speed_ms,0,0.000)
    |   movel(p[0.465113, -0.062298, -0.000100, 0.000000, -3.141593, 0.000000],accel_mss,speed_ms,0,0.000)
    |   speed_ms    = 0.050
    |   movel(p[0.465113, -0.062298, 0.003000, 0.000000, -3.141593, 0.000000],accel_mss,speed_ms,0,blend_radius_m)
    |   speed_ms    = 1.000
    |   movel(p[0.465113, -0.062298, 0.015000, 0.000000, -3.141593, 0.000000],accel_mss,speed_ms,0,blend_radius_m)
    | 
    |   movel(p[0.459410, -0.043732, 0.015000, 0.000000, -3.141593, 0.000000],accel_mss,speed_ms,0,blend_radius_m)
    | 
    |   movel(p[0.459410, -0.043732, 0.003000, 0.000000, -3.141593, 0.000000],accel_mss,speed_ms,0,blend_radius_m)
    |   speed_ms    = 0.050
    |   movel(p[0.459410, -0.043732, -0.000100, 0.000000, -3.141593, 0.000000],accel_mss,speed_ms,0,blend_radius_m)
    |   speed_ms    = 0.083
    |   movel(p[0.459027, -0.043557, -0.000100, 0.000000, 3.141593, 0.000000],accel_mss,speed_ms,0,0.000)
    |   movel(p[0.458627, -0.042974, -0.000100, 0.000000, -3.141593, 0.000000],accel_mss,speed_ms,0,0.000)
    |   movel(p[0.458455, -0.042559, -0.000100, 0.000000, -3.141593, 0.000000],accel_mss,speed_ms,0,0.000)
    |   movel(p[0.458361, -0.042105, -0.000100, 0.000000, -3.141593, 0.000000],accel_mss,speed_ms,0,0.000)
    |   movel(p[0.458356, -0.041736, -0.000100, 0.000000, -3.141593, 0.000000],accel_mss,speed_ms,0,0.000)
    |   movel(p[0.458473, -0.041629, -0.000100, 0.000000, -3.141593, 0.000000],accel_mss,speed_ms,0,0.000)
    |   movel(p[0.458686, -0.041719, -0.000100, 0.000000, -3.141593, 0.000000],accel_mss,speed_ms,0,0.000)
    |   movel(p[0.459026, -0.042107, -0.000100, 0.000000, -3.141593, 0.000000],accel_mss,speed_ms,0,0.000)
    |   movel(p[0.459343, -0.042562, -0.000100, 0.000000, -3.141593, 0.000000],accel_mss,speed_ms,0,0.000)
    |   movel(p[0.459532, -0.042969, -0.000100, 0.000000, -3.141593, 0.000000],accel_mss,speed_ms,0,0.000)
    |   movel(p[0.459618, -0.043527, -0.000100, 0.000000, -3.141593, 0.000000],accel_mss,speed_ms,0,0.000)
    |   movel(p[0.459410, -0.043732, -0.000100, 0.000000, -3.141593, 0.000000],accel_mss,speed_ms,0,0.000)
    |   speed_ms    = 0.050
    |   movel(p[0.459410, -0.043732, 0.003000, 0.000000, -3.141593, 0.000000],accel_mss,speed_ms,0,blend_radius_m)
    |   speed_ms    = 1.000
    |   movel(p[0.459410, -0.043732, 0.015000, 0.000000, -3.141593, 0.000000],accel_mss,speed_ms,0,blend_radius_m)
    | 
    |   movel(p[0.455190, -0.045930, 0.015000, 0.000000, -3.141593, 0.000000],accel_mss,speed_ms,0,blend_radius_m)
    | 
    |   movel(p[0.455190, -0.045930, 0.003000, 0.000000, -3.141593, 0.000000],accel_mss,speed_ms,0,blend_radius_m)
    |   speed_ms    = 0.050
    |   movel(p[0.455190, -0.045930, -0.000100, 0.000000, -3.141593, 0.000000],accel_mss,speed_ms,0,blend_radius_m)
    |   speed_ms    = 0.083
    |   movel(p[0.455112, -0.046492, -0.000100, 0.000000, 3.141593, 0.000000],accel_mss,speed_ms,0,0.000)
    |   movel(p[0.454963, -0.047164, -0.000100, 0.000000, 3.141593, 0.000000],accel_mss,speed_ms,0,0.000)
    |   movel(p[0.454748, -0.047854, -0.000100, 0.000000, 3.141593, 0.000000],accel_mss,speed_ms,0,0.000)
    |   movel(p[0.454638, -0.048174, -0.000100, 0.000000, -3.141593, 0.000000],accel_mss,speed_ms,0,0.000)
    |   movel(p[0.454531, -0.048516, -0.000100, 0.000000, -3.141593, 0.000000],accel_mss,speed_ms,0,0.000)
    |   movel(p[0.454440, -0.048830, -0.000100, 0.000000, -3.141593, 0.000000],accel_mss,speed_ms,0,0.000)
    |   movel(p[0.454385, -0.049054, -0.000100, 0.000000, -3.141593, 0.000000],accel_mss,speed_ms,0,0.000)
    |   movel(p[0.454311, -0.049303, -0.000100, 0.000000, 3.141593, 0.000000],accel_mss,speed_ms,0,0.000)
    |   movel(p[0.454135, -0.049739, -0.000100, 0.000000, -3.141593, 0.000000],accel_mss,speed_ms,0,0.000)
    |   movel(p[0.453913, -0.050242, -0.000100, 0.000000, -3.141593, 0.000000],accel_mss,speed_ms,0,0.000)
    |   movel(p[0.453668, -0.050753, -0.000100, 0.000000, -3.141593, 0.000000],accel_mss,speed_ms,0,0.000)
    |   movel(p[0.453280, -0.051463, -0.000100, 0.000000, -3.141593, 0.000000],accel_mss,speed_ms,0,0.000)
    |   movel(p[0.452899, -0.052018, -0.000100, 0.000000, -3.141593, 0.000000],accel_mss,speed_ms,0,0.000)
    |   movel(p[0.452404, -0.052581, -0.000100, 0.000000, -3.141593, 0.000000],accel_mss,speed_ms,0,0.000)
    |   movel(p[0.451631, -0.053340, -0.000100, 0.000000, -3.141593, 0.000000],accel_mss,speed_ms,0,0.000)
    |   movel(p[0.451079, -0.053853, -0.000100, 0.000000, -3.141593, 0.000000],accel_mss,speed_ms,0,0.000)
    |   movel(p[0.450591, -0.054286, -0.000100, 0.000000, -3.141593, 0.000000],accel_mss,speed_ms,0,0.000)
    |   movel(p[0.450168, -0.054645, -0.000100, 0.000000, -3.141593, 0.000000],accel_mss,speed_ms,0,0.000)
    |   movel(p[0.449987, -0.054694, -0.000100, 0.000000, -3.141593, 0.000000],accel_mss,speed_ms,0,0.000)
    |   movel(p[0.449769, -0.054772, -0.000100, 0.000000, -3.141593, 0.000000],accel_mss,speed_ms,0,0.000)
    |   movel(p[0.449510, -0.054874, -0.000100, 0.000000, 3.141593, 0.000000],accel_mss,speed_ms,0,0.000)
    |   movel(p[0.449230, -0.054995, -0.000100, 0.000000, -3.141593, 0.000000],accel_mss,speed_ms,0,0.000)
    |   movel(p[0.448172, -0.055459, -0.000100, 0.000000, -3.141593, 0.000000],accel_mss,speed_ms,0,0.000)
    |   movel(p[0.447535, -0.055705, -0.000100, 0.000000, -3.141593, 0.000000],accel_mss,speed_ms,0,0.000)
    |   movel(p[0.447016, -0.055853, -0.000100, 0.000000, -3.141593, 0.000000],accel_mss,speed_ms,0,0.000)
    |   movel(p[0.446426, -0.055963, -0.000100, 0.000000, -3.141593, 0.000000],accel_mss,speed_ms,0,0.000)
    |   movel(p[0.446246, -0.055990, -0.000100, 0.000000, -3.141593, 0.000000],accel_mss,speed_ms,0,0.000)
    |   movel(p[0.445872, -0.056050, -0.000100, 0.000000, 3.141593, 0.000000],accel_mss,speed_ms,0,0.000)
    |   movel(p[0.445431, -0.056121, -0.000100, 0.000000, -3.141593, 0.000000],accel_mss,speed_ms,0,0.000)
    |   movel(p[0.444964, -0.056198, -0.000100, 0.000000, -3.141593, 0.000000],accel_mss,speed_ms,0,0.000)
    |   movel(p[0.444284, -0.056288, -0.000100, 0.000000, -3.141593, 0.000000],accel_mss,speed_ms,0,0.000)
    |   movel(p[0.443743, -0.056311, -0.000100, 0.000000, -3.141593, 0.000000],accel_mss,speed_ms,0,0.000)
    |   movel(p[0.443157, -0.056270, -0.000100, 0.000000, -3.141593, 0.000000],accel_mss,speed_ms,0,0.000)
    |   movel(p[0.442313, -0.056149, -0.000100, 0.000000, -3.141593, 0.000000],accel_mss,speed_ms,0,0.000)
    |   movel(p[0.441680, -0.056033, -0.000100, 0.000000, -3.141593, 0.000000],accel_mss,speed_ms,0,0.000)
    |   movel(p[0.441130, -0.055900, -0.000100, 0.000000, 3.141593, 0.000000],accel_mss,speed_ms,0,0.000)
    |   movel(p[0.440693, -0.055761, -0.000100, 0.000000, 3.141593, 0.000000],accel_mss,speed_ms,0,0.000)
    |   movel(p[0.440452, -0.055632, -0.000100, 0.000000, -3.141593, 0.000000],accel_mss,speed_ms,0,0.000)
    |   movel(p[0.440312, -0.055523, -0.000100, 0.000000, -3.141593, 0.000000],accel_mss,speed_ms,0,0.000)
    |   movel(p[0.440200, -0.055424, -0.000100, 0.000000, -3.141593, 0.000000],accel_mss,speed_ms,0,0.000)
    |   movel(p[0.440116, -0.055342, -0.000100, 0.000000, -3.141593, 0.000000],accel_mss,speed_ms,0,0.000)
    |   movel(p[0.440358, -0.055329, -0.000100, 0.000000, -3.141593, 0.000000],accel_mss,speed_ms,0,0.000)
    |   movel(p[0.440604, -0.055365, -0.000100, 0.000000, -3.141593, 0.000000],accel_mss,speed_ms,0,0.000)
    |   movel(p[0.440889, -0.055415, -0.000100, 0.000000, -3.141593, 0.000000],accel_mss,speed_ms,0,0.000)
    |   movel(p[0.442496, -0.055513, -0.000100, 0.000000, -3.141593, 0.000000],accel_mss,speed_ms,0,0.001)
    |   movel(p[0.444504, -0.055260, -0.000100, 0.000000, 3.141593, 0.000000],accel_mss,speed_ms,0,0.001)
    |   movel(p[0.446499, -0.054748, -0.000100, 0.000000, -3.141593, 0.000000],accel_mss,speed_ms,0,0.001)
    |   movel(p[0.448076, -0.054044, -0.000100, 0.000000, -3.141593, 0.000000],accel_mss,speed_ms,0,0.001)
    |   movel(p[0.448236, -0.053955, -0.000100, 0.000000, 3.141593, 0.000000],accel_mss,speed_ms,0,0.000)
    |   movel(p[0.448493, -0.053818, -0.000100, 0.000000, -3.141593, 0.000000],accel_mss,speed_ms,0,0.000)
    |   movel(p[0.448786, -0.053665, -0.000100, 0.000000, 3.141593, 0.000000],accel_mss,speed_ms,0,0.000)
    |   movel(p[0.449076, -0.053517, -0.000100, 0.000000, 3.141593, 0.000000],accel_mss,speed_ms,0,0.000)
    |   movel(p[0.449357, -0.053366, -0.000100, 0.000000, -3.141593, 0.000000],accel_mss,speed_ms,0,0.000)
    |   movel(p[0.449623, -0.053204, -0.000100, 0.000000, -3.141593, 0.000000],accel_mss,speed_ms,0,0.000)
    |   movel(p[0.449844, -0.053053, -0.000100, 0.000000, -3.141593, 0.000000],accel_mss,speed_ms,0,0.000)
    |   movel(p[0.449957, -0.052947, -0.000100, 0.000000, -3.141593, 0.000000],accel_mss,speed_ms,0,0.000)
    |   movel(p[0.450039, -0.052863, -0.000100, 0.000000, -3.141593, 0.000000],accel_mss,speed_ms,0,0.000)
    |   movel(p[0.450135, -0.052793, -0.000100, 0.000000, -3.141593, 0.000000],accel_mss,speed_ms,0,0.000)
    |   movel(p[0.450232, -0.052744, -0.000100, 0.000000, -3.141593, 0.000000],accel_mss,speed_ms,0,0.000)
    |   movel(p[0.450545, -0.052636, -0.000100, 0.000000, -3.141593, 0.000000],accel_mss,speed_ms,0,0.000)
    |   movel(p[0.451271, -0.051930, -0.000100, 0.000000, 3.141593, 0.000000],accel_mss,speed_ms,0,0.000)
    |   movel(p[0.451949, -0.051220, -0.000100, 0.000000, 3.141593, 0.000000],accel_mss,speed_ms,0,0.000)
    |   movel(p[0.452284, -0.050759, -0.000100, 0.000000, 3.141593, 0.000000],accel_mss,speed_ms,0,0.000)
    |   movel(p[0.452372, -0.050601, -0.000100, 0.000000, -3.141593, 0.000000],accel_mss,speed_ms,0,0.000)
    |   movel(p[0.452469, -0.050418, -0.000100, 0.000000, -3.141593, 0.000000],accel_mss,speed_ms,0,0.000)
    |   movel(p[0.452560, -0.050240, -0.000100, 0.000000, 3.141593, 0.000000],accel_mss,speed_ms,0,0.000)
    |   movel(p[0.452629, -0.050098, -0.000100, 0.000000, -3.141593, 0.000000],accel_mss,speed_ms,0,0.000)
    |   movel(p[0.452700, -0.049966, -0.000100, 0.000000, -3.141593, 0.000000],accel_mss,speed_ms,0,0.000)
    |   movel(p[0.452799, -0.049823, -0.000100, 0.000000, -3.141593, 0.000000],accel_mss,speed_ms,0,0.000)
    |   movel(p[0.452908, -0.049690, -0.000100, 0.000000, -3.141593, 0.000000],accel_mss,speed_ms,0,0.000)
    |   movel(p[0.453010, -0.049592, -0.000100, 0.000000, -3.141593, 0.000000],accel_mss,speed_ms,0,0.000)
    |   movel(p[0.453102, -0.049495, -0.000100, 0.000000, -3.141593, 0.000000],accel_mss,speed_ms,0,0.000)
    |   movel(p[0.453180, -0.049371, -0.000100, 0.000000, -3.141593, 0.000000],accel_mss,speed_ms,0,0.000)
    |   movel(p[0.453233, -0.049238, -0.000100, 0.000000, -3.141593, 0.000000],accel_mss,speed_ms,0,0.000)
    |   movel(p[0.453251, -0.049119, -0.000100, 0.000000, -3.141593, 0.000000],accel_mss,speed_ms,0,0.000)
    |   movel(p[0.453261, -0.049008, -0.000100, 0.000000, -3.141593, 0.000000],accel_mss,speed_ms,0,0.000)
    |   movel(p[0.453294, -0.048900, -0.000100, 0.000000, 3.141593, 0.000000],accel_mss,speed_ms,0,0.000)
    |   movel(p[0.453341, -0.048811, -0.000100, 0.000000, -3.141593, 0.000000],accel_mss,speed_ms,0,0.000)
    |   movel(p[0.453477, -0.048676, -0.000100, 0.000000, -3.141593, 0.000000],accel_mss,speed_ms,0,0.000)
    |   movel(p[0.453667, -0.048358, -0.000100, 0.000000, -3.141593, 0.000000],accel_mss,speed_ms,0,0.000)
    |   movel(p[0.453882, -0.047970, -0.000100, 0.000000, -3.141593, 0.000000],accel_mss,speed_ms,0,0.000)
    |   movel(p[0.454109, -0.047527, -0.000100, 0.000000, -3.141593, 0.000000],accel_mss,speed_ms,0,0.000)
    |   movel(p[0.454651, -0.046443, -0.000100, 0.000000, -3.141593, 0.000000],accel_mss,speed_ms,0,0.000)
    |   movel(p[0.454858, -0.046063, -0.000100, 0.000000, -3.141593, 0.000000],accel_mss,speed_ms,0,0.000)
    |   movel(p[0.454987, -0.045881, -0.000100, 0.000000, -3.141593, 0.000000],accel_mss,speed_ms,0,0.000)
    |   movel(p[0.455099, -0.045829, -0.000100, 0.000000, -3.141593, 0.000000],accel_mss,speed_ms,0,0.000)
    |   movel(p[0.455190, -0.045930, -0.000100, 0.000000, -3.141593, 0.000000],accel_mss,speed_ms,0,0.000)
    |   speed_ms    = 0.050
    |   movel(p[0.455190, -0.045930, 0.003000, 0.000000, -3.141593, 0.000000],accel_mss,speed_ms,0,blend_radius_m)
    |   speed_ms    = 1.000
    |   movel(p[0.455190, -0.045930, 0.015000, 0.000000, -3.141593, 0.000000],accel_mss,speed_ms,0,blend_radius_m)
    | 
    |   movel(p[0.457053, -0.043985, 0.015000, 0.000000, -3.141593, 0.000000],accel_mss,speed_ms,0,blend_radius_m)
    | 
    |   movel(p[0.457053, -0.043985, 0.003000, 0.000000, -3.141593, 0.000000],accel_mss,speed_ms,0,blend_radius_m)
    |   speed_ms    = 0.050
    |   movel(p[0.457053, -0.043985, -0.000100, 0.000000, -3.141593, 0.000000],accel_mss,speed_ms,0,blend_radius_m)
    |   speed_ms    = 0.083
    |   movel(p[0.457001, -0.043879, -0.000100, 0.000000, -3.141593, 0.000000],accel_mss,speed_ms,0,0.000)
    |   movel(p[0.457065, -0.043773, -0.000100, 0.000000, -3.141593, 0.000000],accel_mss,speed_ms,0,0.000)
    |   movel(p[0.457219, -0.043729, -0.000100, 0.000000, -3.141593, 0.000000],accel_mss,speed_ms,0,0.000)
    |   movel(p[0.457502, -0.043784, -0.000100, 0.000000, 3.141593, 0.000000],accel_mss,speed_ms,0,0.000)
    |   movel(p[0.457966, -0.043994, -0.000100, 0.000000, 3.141593, 0.000000],accel_mss,speed_ms,0,0.000)
    |   movel(p[0.458417, -0.044237, -0.000100, 0.000000, -3.141593, 0.000000],accel_mss,speed_ms,0,0.000)
    |   movel(p[0.458497, -0.044371, -0.000100, 0.000000, -3.141593, 0.000000],accel_mss,speed_ms,0,0.000)
    |   movel(p[0.458418, -0.044520, -0.000100, 0.000000, 3.141593, 0.000000],accel_mss,speed_ms,0,0.000)
    |   movel(p[0.458217, -0.044576, -0.000100, 0.000000, 3.141593, 0.000000],accel_mss,speed_ms,0,0.000)
    |   movel(p[0.457944, -0.044513, -0.000100, 0.000000, -3.141593, 0.000000],accel_mss,speed_ms,0,0.000)
    |   movel(p[0.457696, -0.044348, -0.000100, 0.000000, -3.141593, 0.000000],accel_mss,speed_ms,0,0.000)
    |   movel(p[0.457553, -0.044226, -0.000100, 0.000000, 3.141593, 0.000000],accel_mss,speed_ms,0,0.000)
    |   movel(p[0.457404, -0.044123, -0.000100, 0.000000, -3.141593, 0.000000],accel_mss,speed_ms,0,0.000)
    |   movel(p[0.457269, -0.044049, -0.000100, 0.000000, -3.141593, 0.000000],accel_mss,speed_ms,0,0.000)
    |   movel(p[0.457111, -0.044018, -0.000100, 0.000000, -3.141593, 0.000000],accel_mss,speed_ms,0,0.000)
    |   speed_ms    = 0.050
    |   movel(p[0.457053, -0.043985, 0.003000, 0.000000, -3.141593, 0.000000],accel_mss,speed_ms,0,blend_radius_m)
    |   speed_ms    = 1.000
    |   movel(p[0.457053, -0.043985, 0.015000, 0.000000, -3.141593, 0.000000],accel_mss,speed_ms,0,blend_radius_m)
    | 
    |   movel(p[0.451490, -0.046380, 0.015000, 0.000000, 3.141593, 0.000000],accel_mss,speed_ms,0,blend_radius_m)
    | 
    |   movel(p[0.451490, -0.046380, 0.003000, 0.000000, -3.141593, 0.000000],accel_mss,speed_ms,0,blend_radius_m)
    |   speed_ms    = 0.050
    |   movel(p[0.451490, -0.046380, -0.000100, 0.000000, -3.141593, 0.000000],accel_mss,speed_ms,0,blend_radius_m)
    |   speed_ms    = 0.083
    |   movel(p[0.451577, -0.046592, -0.000100, 0.000000, -3.141593, 0.000000],accel_mss,speed_ms,0,0.000)
    |   movel(p[0.451597, -0.046714, -0.000100, 0.000000, 3.141593, 0.000000],accel_mss,speed_ms,0,0.000)
    |   movel(p[0.451472, -0.046847, -0.000100, 0.000000, -3.141593, 0.000000],accel_mss,speed_ms,0,0.000)
    |   movel(p[0.451366, -0.046898, -0.000100, 0.000000, -3.141593, 0.000000],accel_mss,speed_ms,0,0.000)
    |   movel(p[0.451191, -0.047016, -0.000100, 0.000000, 3.141593, 0.000000],accel_mss,speed_ms,0,0.000)
    |   movel(p[0.450994, -0.047165, -0.000100, 0.000000, -3.141593, 0.000000],accel_mss,speed_ms,0,0.000)
    |   movel(p[0.450799, -0.047328, -0.000100, 0.000000, -3.141593, 0.000000],accel_mss,speed_ms,0,0.000)
    |   movel(p[0.450271, -0.047740, -0.000100, 0.000000, -3.141593, 0.000000],accel_mss,speed_ms,0,0.000)
    |   movel(p[0.449712, -0.048078, -0.000100, 0.000000, 3.141593, 0.000000],accel_mss,speed_ms,0,0.000)
    |   movel(p[0.449192, -0.048308, -0.000100, 0.000000, 3.141593, 0.000000],accel_mss,speed_ms,0,0.000)
    |   movel(p[0.448793, -0.048379, -0.000100, 0.000000, -3.141593, 0.000000],accel_mss,speed_ms,0,0.000)
    |   movel(p[0.448615, -0.048355, -0.000100, 0.000000, -3.141593, 0.000000],accel_mss,speed_ms,0,0.000)
    |   movel(p[0.448410, -0.048283, -0.000100, 0.000000, -3.141593, 0.000000],accel_mss,speed_ms,0,0.000)
    |   movel(p[0.448210, -0.048178, -0.000100, 0.000000, -3.141593, 0.000000],accel_mss,speed_ms,0,0.000)
    |   movel(p[0.448048, -0.048053, -0.000100, 0.000000, -3.141593, 0.000000],accel_mss,speed_ms,0,0.000)
    |   movel(p[0.447839, -0.047788, -0.000100, 0.000000, 3.141593, 0.000000],accel_mss,speed_ms,0,0.000)
    |   movel(p[0.447709, -0.047465, -0.000100, 0.000000, -3.141593, 0.000000],accel_mss,speed_ms,0,0.000)
    |   movel(p[0.447730, -0.047283, -0.000100, 0.000000, -3.141593, 0.000000],accel_mss,speed_ms,0,0.000)
    |   movel(p[0.447846, -0.047251, -0.000100, 0.000000, -3.141593, 0.000000],accel_mss,speed_ms,0,0.000)
    |   movel(p[0.448036, -0.047270, -0.000100, 0.000000, -3.141593, 0.000000],accel_mss,speed_ms,0,0.000)
    |   movel(p[0.448548, -0.047064, -0.000100, 0.000000, -3.141593, 0.000000],accel_mss,speed_ms,0,0.000)
    |   movel(p[0.449172, -0.046758, -0.000100, 0.000000, -3.141593, 0.000000],accel_mss,speed_ms,0,0.000)
    |   movel(p[0.449876, -0.046356, -0.000100, 0.000000, -3.141593, 0.000000],accel_mss,speed_ms,0,0.000)
    |   movel(p[0.450443, -0.046073, -0.000100, 0.000000, -3.141593, 0.000000],accel_mss,speed_ms,0,0.000)
    |   movel(p[0.450903, -0.045988, -0.000100, 0.000000, -3.141593, 0.000000],accel_mss,speed_ms,0,0.000)
    |   movel(p[0.451250, -0.046097, -0.000100, 0.000000, 3.141593, 0.000000],accel_mss,speed_ms,0,0.000)
    |   movel(p[0.451490, -0.046380, -0.000100, 0.000000, -3.141593, 0.000000],accel_mss,speed_ms,0,0.000)
    |   speed_ms    = 0.050
    |   movel(p[0.451490, -0.046380, 0.003000, 0.000000, -3.141593, 0.000000],accel_mss,speed_ms,0,blend_radius_m)
    |   speed_ms    = 1.000
    |   movel(p[0.451490, -0.046380, 0.015000, 0.000000, 3.141593, 0.000000],accel_mss,speed_ms,0,blend_radius_m)
    | 
    |   movel(p[0.383835, -0.046267, 0.015000, 0.000000, -3.141593, 0.000000],accel_mss,speed_ms,0,blend_radius_m)
    | 
    |   movel(p[0.383835, -0.046267, 0.003000, 0.000000, 3.141593, 0.000000],accel_mss,speed_ms,0,blend_radius_m)
    |   speed_ms    = 0.050
    |   movel(p[0.383835, -0.046267, -0.000100, 0.000000, -3.141593, 0.000000],accel_mss,speed_ms,0,blend_radius_m)
    |   speed_ms    = 0.083
    |   movel(p[0.383686, -0.047704, -0.000100, 0.000000, -3.141593, 0.000000],accel_mss,speed_ms,0,0.001)
    |   movel(p[0.383613, -0.048161, -0.000100, 0.000000, -3.141593, 0.000000],accel_mss,speed_ms,0,0.000)
    |   movel(p[0.383537, -0.048666, -0.000100, 0.000000, -3.141593, 0.000000],accel_mss,speed_ms,0,0.000)
    |   movel(p[0.383468, -0.049143, -0.000100, 0.000000, -3.141593, 0.000000],accel_mss,speed_ms,0,0.000)
    |   movel(p[0.383420, -0.049504, -0.000100, 0.000000, 3.141593, 0.000000],accel_mss,speed_ms,0,0.000)
    |   movel(p[0.383362, -0.049870, -0.000100, 0.000000, -3.141593, 0.000000],accel_mss,speed_ms,0,0.000)
    |   movel(p[0.383263, -0.050364, -0.000100, 0.000000, 3.141593, 0.000000],accel_mss,speed_ms,0,0.000)
    |   movel(p[0.383144, -0.050893, -0.000100, 0.000000, 3.141593, 0.000000],accel_mss,speed_ms,0,0.000)
    |   movel(p[0.383020, -0.051379, -0.000100, 0.000000, -3.141593, 0.000000],accel_mss,speed_ms,0,0.000)
    |   movel(p[0.382884, -0.051882, -0.000100, 0.000000, -3.141593, 0.000000],accel_mss,speed_ms,0,0.000)
    |   movel(p[0.382727, -0.052465, -0.000100, 0.000000, -3.141593, 0.000000],accel_mss,speed_ms,0,0.000)
    |   movel(p[0.382574, -0.053035, -0.000100, 0.000000, 3.141593, 0.000000],accel_mss,speed_ms,0,0.000)
    |   movel(p[0.382452, -0.053496, -0.000100, 0.000000, -3.141593, 0.000000],accel_mss,speed_ms,0,0.000)
    |   movel(p[0.382199, -0.054369, -0.000100, 0.000000, -3.141593, 0.000000],accel_mss,speed_ms,0,0.000)
    |   movel(p[0.381783, -0.055658, -0.000100, 0.000000, -3.141593, 0.000000],accel_mss,speed_ms,0,0.001)
    |   movel(p[0.381355, -0.056922, -0.000100, 0.000000, -3.141593, 0.000000],accel_mss,speed_ms,0,0.001)
    |   movel(p[0.381091, -0.057604, -0.000100, 0.000000, 3.141593, 0.000000],accel_mss,speed_ms,0,0.000)
    |   movel(p[0.381014, -0.057791, -0.000100, 0.000000, -3.141593, 0.000000],accel_mss,speed_ms,0,0.000)
    |   movel(p[0.380845, -0.058220, -0.000100, 0.000000, 3.141593, 0.000000],accel_mss,speed_ms,0,0.000)
    |   movel(p[0.380646, -0.058731, -0.000100, 0.000000, 3.141593, 0.000000],accel_mss,speed_ms,0,0.000)
    |   movel(p[0.380435, -0.059280, -0.000100, 0.000000, 3.141593, 0.000000],accel_mss,speed_ms,0,0.000)
    |   movel(p[0.380204, -0.059871, -0.000100, 0.000000, -3.141593, 0.000000],accel_mss,speed_ms,0,0.000)
    |   movel(p[0.379949, -0.060508, -0.000100, 0.000000, -3.141593, 0.000000],accel_mss,speed_ms,0,0.000)
    |   movel(p[0.379705, -0.061099, -0.000100, 0.000000, -3.141593, 0.000000],accel_mss,speed_ms,0,0.000)
    |   movel(p[0.379520, -0.061530, -0.000100, 0.000000, -3.141593, 0.000000],accel_mss,speed_ms,0,0.000)
    |   movel(p[0.379363, -0.061886, -0.000100, 0.000000, -3.141593, 0.000000],accel_mss,speed_ms,0,0.000)
    |   movel(p[0.379209, -0.062235, -0.000100, 0.000000, -3.141593, 0.000000],accel_mss,speed_ms,0,0.000)
    |   movel(p[0.379076, -0.062535, -0.000100, 0.000000, -3.141593, 0.000000],accel_mss,speed_ms,0,0.000)
    |   movel(p[0.379002, -0.062704, -0.000100, 0.000000, -3.141593, 0.000000],accel_mss,speed_ms,0,0.000)
    |   movel(p[0.378934, -0.062859, -0.000100, 0.000000, -3.141593, 0.000000],accel_mss,speed_ms,0,0.000)
    |   movel(p[0.378831, -0.063091, -0.000100, 0.000000, -3.141593, 0.000000],accel_mss,speed_ms,0,0.000)
    |   movel(p[0.378715, -0.063350, -0.000100, 0.000000, -3.141593, 0.000000],accel_mss,speed_ms,0,0.000)
    |   movel(p[0.378602, -0.063601, -0.000100, 0.000000, -3.141593, 0.000000],accel_mss,speed_ms,0,0.000)
    |   movel(p[0.378468, -0.063900, -0.000100, 0.000000, -3.141593, 0.000000],accel_mss,speed_ms,0,0.000)
    |   movel(p[0.378334, -0.064198, -0.000100, 0.000000, 3.141593, 0.000000],accel_mss,speed_ms,0,0.000)
    |   movel(p[0.378174, -0.063262, -0.000100, 0.000000, -3.141593, 0.000000],accel_mss,speed_ms,0,0.000)
    |   movel(p[0.378014, -0.062326, -0.000100, 0.000000, -3.141593, 0.000000],accel_mss,speed_ms,0,0.000)
    |   movel(p[0.377706, -0.060662, -0.000100, 0.000000, -3.141593, 0.000000],accel_mss,speed_ms,0,0.001)
    |   movel(p[0.377415, -0.059414, -0.000100, 0.000000, -3.141593, 0.000000],accel_mss,speed_ms,0,0.001)
    |   movel(p[0.377137, -0.058510, -0.000100, 0.000000, 3.141593, 0.000000],accel_mss,speed_ms,0,0.000)
    |   movel(p[0.376876, -0.058061, -0.000100, 0.000000, -3.141593, 0.000000],accel_mss,speed_ms,0,0.000)
    |   movel(p[0.376787, -0.057907, -0.000100, 0.000000, -3.141593, 0.000000],accel_mss,speed_ms,0,0.000)
    |   movel(p[0.376751, -0.057734, -0.000100, 0.000000, -3.141593, 0.000000],accel_mss,speed_ms,0,0.000)
    |   movel(p[0.376634, -0.057233, -0.000100, 0.000000, -3.141593, 0.000000],accel_mss,speed_ms,0,0.000)
    |   movel(p[0.376018, -0.056033, -0.000100, 0.000000, -3.141593, 0.000000],accel_mss,speed_ms,0,0.001)
    |   movel(p[0.375351, -0.054865, -0.000100, 0.000000, -3.141593, 0.000000],accel_mss,speed_ms,0,0.001)
    |   movel(p[0.374862, -0.054221, -0.000100, 0.000000, -3.141593, 0.000000],accel_mss,speed_ms,0,0.000)
    |   movel(p[0.374724, -0.054063, -0.000100, 0.000000, -3.141593, 0.000000],accel_mss,speed_ms,0,0.000)
    |   movel(p[0.374607, -0.053908, -0.000100, 0.000000, -3.141593, 0.000000],accel_mss,speed_ms,0,0.000)
    |   movel(p[0.374521, -0.053771, -0.000100, 0.000000, -3.141593, 0.000000],accel_mss,speed_ms,0,0.000)
    |   movel(p[0.374413, -0.053481, -0.000100, 0.000000, -3.141593, 0.000000],accel_mss,speed_ms,0,0.000)
    |   movel(p[0.372964, -0.052020, -0.000100, 0.000000, -3.141593, 0.000000],accel_mss,speed_ms,0,0.001)
    |   movel(p[0.371506, -0.050566, -0.000100, 0.000000, -3.141593, 0.000000],accel_mss,speed_ms,0,0.001)
    |   movel(p[0.371295, -0.050479, -0.000100, 0.000000, -3.141593, 0.000000],accel_mss,speed_ms,0,0.000)
    |   movel(p[0.371035, -0.050344, -0.000100, 0.000000, -3.141593, 0.000000],accel_mss,speed_ms,0,0.000)
    |   movel(p[0.370819, -0.050195, -0.000100, 0.000000, 3.141593, 0.000000],accel_mss,speed_ms,0,0.000)
    |   movel(p[0.370587, -0.050019, -0.000100, 0.000000, -3.141593, 0.000000],accel_mss,speed_ms,0,0.000)
    |   movel(p[0.369617, -0.049385, -0.000100, 0.000000, -3.141593, 0.000000],accel_mss,speed_ms,0,0.000)
    |   movel(p[0.368053, -0.048613, -0.000100, 0.000000, -3.141593, 0.000000],accel_mss,speed_ms,0,0.001)
    |   movel(p[0.366393, -0.047911, -0.000100, 0.000000, -3.141593, 0.000000],accel_mss,speed_ms,0,0.001)
    |   movel(p[0.365051, -0.047480, -0.000100, 0.000000, -3.141593, 0.000000],accel_mss,speed_ms,0,0.001)
    |   movel(p[0.363794, -0.047171, -0.000100, 0.000000, -3.141593, 0.000000],accel_mss,speed_ms,0,0.001)
    |   movel(p[0.362941, -0.046997, -0.000100, 0.000000, -3.141593, 0.000000],accel_mss,speed_ms,0,0.000)
    |   movel(p[0.362138, -0.046883, -0.000100, 0.000000, -3.141593, 0.000000],accel_mss,speed_ms,0,0.000)
    |   movel(p[0.361079, -0.046785, -0.000100, 0.000000, -3.141593, 0.000000],accel_mss,speed_ms,0,0.000)
    |   movel(p[0.360670, -0.046749, -0.000100, 0.000000, -3.141593, 0.000000],accel_mss,speed_ms,0,0.000)
    |   movel(p[0.360306, -0.046707, -0.000100, 0.000000, -3.141593, 0.000000],accel_mss,speed_ms,0,0.000)
    |   movel(p[0.360002, -0.046664, -0.000100, 0.000000, 3.141593, 0.000000],accel_mss,speed_ms,0,0.000)
    |   movel(p[0.359835, -0.046545, -0.000100, 0.000000, -3.141593, 0.000000],accel_mss,speed_ms,0,0.000)
    |   movel(p[0.359822, -0.046435, -0.000100, 0.000000, 3.141593, 0.000000],accel_mss,speed_ms,0,0.000)
    |   movel(p[0.359884, -0.046250, -0.000100, 0.000000, -3.141593, 0.000000],accel_mss,speed_ms,0,0.000)
    |   movel(p[0.360103, -0.045783, -0.000100, 0.000000, -3.141593, 0.000000],accel_mss,speed_ms,0,0.000)
    |   movel(p[0.360387, -0.045219, -0.000100, 0.000000, -3.141593, 0.000000],accel_mss,speed_ms,0,0.000)
    |   movel(p[0.360625, -0.044811, -0.000100, 0.000000, -3.141593, 0.000000],accel_mss,speed_ms,0,0.000)
    |   movel(p[0.360907, -0.044409, -0.000100, 0.000000, -3.141593, 0.000000],accel_mss,speed_ms,0,0.000)
    |   movel(p[0.361338, -0.043859, -0.000100, 0.000000, -3.141593, 0.000000],accel_mss,speed_ms,0,0.000)
    |   movel(p[0.361554, -0.043582, -0.000100, 0.000000, -3.141593, 0.000000],accel_mss,speed_ms,0,0.000)
    |   movel(p[0.361735, -0.043327, -0.000100, 0.000000, -3.141593, 0.000000],accel_mss,speed_ms,0,0.000)
    |   movel(p[0.361877, -0.043109, -0.000100, 0.000000, -3.141593, 0.000000],accel_mss,speed_ms,0,0.000)
    |   movel(p[0.361926, -0.042946, -0.000100, 0.000000, -3.141593, 0.000000],accel_mss,speed_ms,0,0.000)
    |   movel(p[0.362055, -0.042779, -0.000100, 0.000000, -3.141593, 0.000000],accel_mss,speed_ms,0,0.000)
    |   movel(p[0.362225, -0.042584, -0.000100, 0.000000, -3.141593, 0.000000],accel_mss,speed_ms,0,0.000)
    |   movel(p[0.362426, -0.042379, -0.000100, 0.000000, -3.141593, 0.000000],accel_mss,speed_ms,0,0.000)
    |   movel(p[0.362627, -0.042172, -0.000100, 0.000000, -3.141593, 0.000000],accel_mss,speed_ms,0,0.000)
    |   movel(p[0.362796, -0.041971, -0.000100, 0.000000, -3.141593, 0.000000],accel_mss,speed_ms,0,0.000)
    |   movel(p[0.362923, -0.041797, -0.000100, 0.000000, -3.141593, 0.000000],accel_mss,speed_ms,0,0.000)
    |   movel(p[0.362982, -0.041610, -0.000100, 0.000000, -3.141593, 0.000000],accel_mss,speed_ms,0,0.000)
    |   movel(p[0.363149, -0.041395, -0.000100, 0.000000, -3.141593, 0.000000],accel_mss,speed_ms,0,0.000)
    |   movel(p[0.363367, -0.041145, -0.000100, 0.000000, -3.141593, 0.000000],accel_mss,speed_ms,0,0.000)
    |   movel(p[0.363626, -0.040879, -0.000100, 0.000000, 3.141593, 0.000000],accel_mss,speed_ms,0,0.000)
    |   movel(p[0.363884, -0.040614, -0.000100, 0.000000, 3.141593, 0.000000],accel_mss,speed_ms,0,0.000)
    |   movel(p[0.364102, -0.040366, -0.000100, 0.000000, 3.141593, 0.000000],accel_mss,speed_ms,0,0.000)
    |   movel(p[0.364270, -0.040153, -0.000100, 0.000000, -3.141593, 0.000000],accel_mss,speed_ms,0,0.000)
    |   movel(p[0.364399, -0.039823, -0.000100, 0.000000, 3.141593, 0.000000],accel_mss,speed_ms,0,0.000)
    |   movel(p[0.365539, -0.038669, -0.000100, 0.000000, 3.141593, 0.000000],accel_mss,speed_ms,0,0.001)
    |   movel(p[0.366692, -0.037527, -0.000100, 0.000000, -3.141593, 0.000000],accel_mss,speed_ms,0,0.001)
    |   movel(p[0.366932, -0.037429, -0.000100, 0.000000, -3.141593, 0.000000],accel_mss,speed_ms,0,0.000)
    |   movel(p[0.367173, -0.037297, -0.000100, 0.000000, -3.141593, 0.000000],accel_mss,speed_ms,0,0.000)
    |   movel(p[0.367349, -0.037151, -0.000100, 0.000000, 3.141593, 0.000000],accel_mss,speed_ms,0,0.000)
    |   movel(p[0.367526, -0.036979, -0.000100, 0.000000, -3.141593, 0.000000],accel_mss,speed_ms,0,0.000)
    |   movel(p[0.367704, -0.036807, -0.000100, 0.000000, -3.141593, 0.000000],accel_mss,speed_ms,0,0.000)
    |   movel(p[0.367883, -0.036661, -0.000100, 0.000000, -3.141593, 0.000000],accel_mss,speed_ms,0,0.000)
    |   movel(p[0.368041, -0.036555, -0.000100, 0.000000, -3.141593, 0.000000],accel_mss,speed_ms,0,0.000)
    |   movel(p[0.368217, -0.036513, -0.000100, 0.000000, 3.141593, 0.000000],accel_mss,speed_ms,0,0.000)
    |   movel(p[0.368316, -0.036464, -0.000100, 0.000000, -3.141593, 0.000000],accel_mss,speed_ms,0,0.000)
    |   movel(p[0.368414, -0.036392, -0.000100, 0.000000, 3.141593, 0.000000],accel_mss,speed_ms,0,0.000)
    |   movel(p[0.368498, -0.036307, -0.000100, 0.000000, -3.141593, 0.000000],accel_mss,speed_ms,0,0.000)
    |   movel(p[0.368596, -0.036208, -0.000100, 0.000000, -3.141593, 0.000000],accel_mss,speed_ms,0,0.000)
    |   movel(p[0.368745, -0.036091, -0.000100, 0.000000, 3.141593, 0.000000],accel_mss,speed_ms,0,0.000)
    |   movel(p[0.368914, -0.035976, -0.000100, 0.000000, -3.141593, 0.000000],accel_mss,speed_ms,0,0.000)
    |   movel(p[0.369079, -0.035882, -0.000100, 0.000000, 3.141593, 0.000000],accel_mss,speed_ms,0,0.000)
    |   movel(p[0.369268, -0.035782, -0.000100, 0.000000, 3.141593, 0.000000],accel_mss,speed_ms,0,0.000)
    |   movel(p[0.369513, -0.035650, -0.000100, 0.000000, -3.141593, 0.000000],accel_mss,speed_ms,0,0.000)
    |   movel(p[0.369771, -0.035507, -0.000100, 0.000000, -3.141593, 0.000000],accel_mss,speed_ms,0,0.000)
    |   movel(p[0.370001, -0.035378, -0.000100, 0.000000, -3.141593, 0.000000],accel_mss,speed_ms,0,0.000)
    |   movel(p[0.370902, -0.034937, -0.000100, 0.000000, -3.141593, 0.000000],accel_mss,speed_ms,0,0.000)
    |   movel(p[0.371836, -0.034629, -0.000100, 0.000000, -3.141593, 0.000000],accel_mss,speed_ms,0,0.000)
    |   movel(p[0.372828, -0.034447, -0.000100, 0.000000, -3.141593, 0.000000],accel_mss,speed_ms,0,0.000)
    |   movel(p[0.373901, -0.034384, -0.000100, 0.000000, -3.141593, 0.000000],accel_mss,speed_ms,0,0.000)
    |   movel(p[0.375046, -0.034438, -0.000100, 0.000000, -3.141593, 0.000000],accel_mss,speed_ms,0,0.000)
    |   movel(p[0.376045, -0.034606, -0.000100, 0.000000, -3.141593, 0.000000],accel_mss,speed_ms,0,0.000)
    |   movel(p[0.376998, -0.034912, -0.000100, 0.000000, -3.141593, 0.000000],accel_mss,speed_ms,0,0.000)
    |   movel(p[0.378001, -0.035379, -0.000100, 0.000000, -3.141593, 0.000000],accel_mss,speed_ms,0,0.000)
    |   movel(p[0.378827, -0.035824, -0.000100, 0.000000, -3.141593, 0.000000],accel_mss,speed_ms,0,0.000)
    |   movel(p[0.379236, -0.036063, -0.000100, 0.000000, -3.141593, 0.000000],accel_mss,speed_ms,0,0.000)
    |   movel(p[0.379518, -0.036262, -0.000100, 0.000000, -3.141593, 0.000000],accel_mss,speed_ms,0,0.000)
    |   movel(p[0.379803, -0.036508, -0.000100, 0.000000, -3.141593, 0.000000],accel_mss,speed_ms,0,0.000)
    |   movel(p[0.379945, -0.036631, -0.000100, 0.000000, -3.141593, 0.000000],accel_mss,speed_ms,0,0.000)
    |   movel(p[0.380087, -0.036735, -0.000100, 0.000000, 3.141593, 0.000000],accel_mss,speed_ms,0,0.000)
    |   movel(p[0.380213, -0.036810, -0.000100, 0.000000, -3.141593, 0.000000],accel_mss,speed_ms,0,0.000)
    |   movel(p[0.380492, -0.036912, -0.000100, 0.000000, -3.141593, 0.000000],accel_mss,speed_ms,0,0.000)
    |   movel(p[0.381412, -0.037835, -0.000100, 0.000000, -3.141593, 0.000000],accel_mss,speed_ms,0,0.001)
    |   movel(p[0.382279, -0.038734, -0.000100, 0.000000, -3.141593, 0.000000],accel_mss,speed_ms,0,0.000)
    |   movel(p[0.382506, -0.039079, -0.000100, 0.000000, 3.141593, 0.000000],accel_mss,speed_ms,0,0.000)
    |   movel(p[0.382563, -0.039198, -0.000100, 0.000000, 3.141593, 0.000000],accel_mss,speed_ms,0,0.000)
    |   movel(p[0.382664, -0.039385, -0.000100, 0.000000, -3.141593, 0.000000],accel_mss,speed_ms,0,0.000)
    |   movel(p[0.382783, -0.039597, -0.000100, 0.000000, -3.141593, 0.000000],accel_mss,speed_ms,0,0.000)
    |   movel(p[0.382906, -0.039805, -0.000100, 0.000000, 3.141593, 0.000000],accel_mss,speed_ms,0,0.000)
    |   movel(p[0.383044, -0.040082, -0.000100, 0.000000, 3.141593, 0.000000],accel_mss,speed_ms,0,0.000)
    |   movel(p[0.383214, -0.040540, -0.000100, 0.000000, 3.141593, 0.000000],accel_mss,speed_ms,0,0.000)
    |   movel(p[0.383384, -0.041071, -0.000100, 0.000000, -3.141593, 0.000000],accel_mss,speed_ms,0,0.000)
    |   movel(p[0.383529, -0.041605, -0.000100, 0.000000, -3.141593, 0.000000],accel_mss,speed_ms,0,0.000)
    |   movel(p[0.383750, -0.042900, -0.000100, 0.000000, -3.141593, 0.000000],accel_mss,speed_ms,0,0.001)
    |   movel(p[0.383852, -0.044562, -0.000100, 0.000000, -3.141593, 0.000000],accel_mss,speed_ms,0,0.001)
    |   movel(p[0.383835, -0.046267, -0.000100, 0.000000, -3.141593, 0.000000],accel_mss,speed_ms,0,0.001)
    |   speed_ms    = 0.050
    |   movel(p[0.383835, -0.046267, 0.003000, 0.000000, 3.141593, 0.000000],accel_mss,speed_ms,0,blend_radius_m)
    |   speed_ms    = 1.000
    |   movel(p[0.383835, -0.046267, 0.015000, 0.000000, -3.141593, 0.000000],accel_mss,speed_ms,0,blend_radius_m)
    | 
    |   movel(p[0.472020, -0.117441, 0.015000, 0.000000, -3.141593, 0.000000],accel_mss,speed_ms,0,blend_radius_m)
    | 
    |   movel(p[0.472020, -0.117441, 0.003000, 0.000000, -3.141593, 0.000000],accel_mss,speed_ms,0,blend_radius_m)
    |   speed_ms    = 0.050
    |   movel(p[0.472020, -0.117441, -0.000100, 0.000000, -3.141593, 0.000000],accel_mss,speed_ms,0,blend_radius_m)
    |   speed_ms    = 0.083
    |   movel(p[0.472756, -0.116567, -0.000100, 0.000000, -3.141593, 0.000000],accel_mss,speed_ms,0,0.000)
    |   movel(p[0.473435, -0.116041, -0.000100, 0.000000, -3.141593, 0.000000],accel_mss,speed_ms,0,0.000)
    |   movel(p[0.474082, -0.115723, -0.000100, 0.000000, -3.141593, 0.000000],accel_mss,speed_ms,0,0.000)
    |   movel(p[0.474875, -0.115540, -0.000100, 0.000000, -3.141593, 0.000000],accel_mss,speed_ms,0,0.000)
    |   movel(p[0.476051, -0.115436, -0.000100, 0.000000, -3.141593, 0.000000],accel_mss,speed_ms,0,0.000)
    |   movel(p[0.476838, -0.115395, -0.000100, 0.000000, -3.141593, 0.000000],accel_mss,speed_ms,0,0.000)
    |   movel(p[0.477626, -0.115354, -0.000100, 0.000000, -3.141593, 0.000000],accel_mss,speed_ms,0,0.000)
    |   movel(p[0.477644, -0.115091, -0.000100, 0.000000, -3.141593, 0.000000],accel_mss,speed_ms,0,0.000)
    |   movel(p[0.477663, -0.114829, -0.000100, 0.000000, -3.141593, 0.000000],accel_mss,speed_ms,0,0.000)
    |   movel(p[0.477683, -0.114563, -0.000100, 0.000000, -3.141593, 0.000000],accel_mss,speed_ms,0,0.000)
    |   movel(p[0.477715, -0.114181, -0.000100, 0.000000, -3.141593, 0.000000],accel_mss,speed_ms,0,0.000)
    |   movel(p[0.477751, -0.113760, -0.000100, 0.000000, -3.141593, 0.000000],accel_mss,speed_ms,0,0.000)
    |   movel(p[0.477788, -0.113360, -0.000100, 0.000000, -3.141593, 0.000000],accel_mss,speed_ms,0,0.000)
    |   movel(p[0.477832, -0.112888, -0.000100, 0.000000, -3.141593, 0.000000],accel_mss,speed_ms,0,0.000)
    |   movel(p[0.477876, -0.112416, -0.000100, 0.000000, -3.141593, 0.000000],accel_mss,speed_ms,0,0.000)
    |   movel(p[0.478413, -0.112438, -0.000100, 0.000000, -3.141593, 0.000000],accel_mss,speed_ms,0,0.000)
    |   movel(p[0.478951, -0.112460, -0.000100, 0.000000, -3.141593, 0.000000],accel_mss,speed_ms,0,0.000)
    |   movel(p[0.479488, -0.112482, -0.000100, 0.000000, -3.141593, 0.000000],accel_mss,speed_ms,0,0.000)
    |   movel(p[0.480026, -0.112504, -0.000100, 0.000000, -3.141593, 0.000000],accel_mss,speed_ms,0,0.000)
    |   movel(p[0.480047, -0.114379, -0.000100, 0.000000, -3.141593, 0.000000],accel_mss,speed_ms,0,0.001)
    |   movel(p[0.480068, -0.116254, -0.000100, 0.000000, -3.141593, 0.000000],accel_mss,speed_ms,0,0.001)
    |   movel(p[0.480078, -0.117716, -0.000100, 0.000000, -3.141593, 0.000000],accel_mss,speed_ms,0,0.001)
    |   movel(p[0.480073, -0.119003, -0.000100, 0.000000, -3.141593, 0.000000],accel_mss,speed_ms,0,0.001)
    |   movel(p[0.480058, -0.120097, -0.000100, 0.000000, -3.141593, 0.000000],accel_mss,speed_ms,0,0.000)
    |   movel(p[0.480026, -0.120348, -0.000100, 0.000000, -3.141593, 0.000000],accel_mss,speed_ms,0,0.000)
    |   movel(p[0.479937, -0.120539, -0.000100, 0.000000, -3.141593, 0.000000],accel_mss,speed_ms,0,0.000)
    |   movel(p[0.479796, -0.120635, -0.000100, 0.000000, -3.141593, 0.000000],accel_mss,speed_ms,0,0.000)
    |   movel(p[0.479528, -0.120667, -0.000100, 0.000000, -3.141593, 0.000000],accel_mss,speed_ms,0,0.000)
    |   movel(p[0.478859, -0.120648, -0.000100, 0.000000, -3.141593, 0.000000],accel_mss,speed_ms,0,0.000)
    |   movel(p[0.478317, -0.120626, -0.000100, 0.000000, -3.141593, 0.000000],accel_mss,speed_ms,0,0.000)
    |   movel(p[0.477776, -0.120604, -0.000100, 0.000000, -3.141593, 0.000000],accel_mss,speed_ms,0,0.000)
    |   movel(p[0.477754, -0.119866, -0.000100, 0.000000, -3.141593, 0.000000],accel_mss,speed_ms,0,0.000)
    |   movel(p[0.477733, -0.119128, -0.000100, 0.000000, -3.141593, 0.000000],accel_mss,speed_ms,0,0.000)
    |   movel(p[0.477711, -0.118389, -0.000100, 0.000000, -3.141593, 0.000000],accel_mss,speed_ms,0,0.000)
    |   movel(p[0.477689, -0.117651, -0.000100, 0.000000, -3.141593, 0.000000],accel_mss,speed_ms,0,0.000)
    |   movel(p[0.476947, -0.117677, -0.000100, 0.000000, -3.141593, 0.000000],accel_mss,speed_ms,0,0.000)
    |   movel(p[0.476205, -0.117703, -0.000100, 0.000000, -3.141593, 0.000000],accel_mss,speed_ms,0,0.000)
    |   movel(p[0.475291, -0.117745, -0.000100, 0.000000, -3.141593, 0.000000],accel_mss,speed_ms,0,0.000)
    |   movel(p[0.474869, -0.117810, -0.000100, 0.000000, -3.141593, 0.000000],accel_mss,speed_ms,0,0.000)
    |   movel(p[0.474577, -0.117940, -0.000100, 0.000000, -3.141593, 0.000000],accel_mss,speed_ms,0,0.000)
    |   movel(p[0.474264, -0.118191, -0.000100, 0.000000, -3.141593, 0.000000],accel_mss,speed_ms,0,0.000)
    |   movel(p[0.473760, -0.118872, -0.000100, 0.000000, -3.141593, 0.000000],accel_mss,speed_ms,0,0.000)
    |   movel(p[0.473547, -0.119643, -0.000100, 0.000000, -3.141593, 0.000000],accel_mss,speed_ms,0,0.000)
    |   movel(p[0.473651, -0.120426, -0.000100, 0.000000, -3.141593, 0.000000],accel_mss,speed_ms,0,0.000)
    |   movel(p[0.474056, -0.121137, -0.000100, 0.000000, -3.141593, 0.000000],accel_mss,speed_ms,0,0.000)
    |   movel(p[0.474235, -0.121328, -0.000100, 0.000000, -3.141593, 0.000000],accel_mss,speed_ms,0,0.000)
    |   movel(p[0.474448, -0.121513, -0.000100, 0.000000, -3.141593, 0.000000],accel_mss,speed_ms,0,0.000)
    |   movel(p[0.474661, -0.121667, -0.000100, 0.000000, -3.141593, 0.000000],accel_mss,speed_ms,0,0.000)
    |   movel(p[0.474837, -0.121759, -0.000100, 0.000000, -3.141593, 0.000000],accel_mss,speed_ms,0,0.000)
    |   movel(p[0.475148, -0.121826, -0.000100, 0.000000, -3.141593, 0.000000],accel_mss,speed_ms,0,0.000)
    |   movel(p[0.476238, -0.121865, -0.000100, 0.000000, -3.141593, 0.000000],accel_mss,speed_ms,0,0.000)
    |   movel(p[0.477626, -0.121888, -0.000100, 0.000000, -3.141593, 0.000000],accel_mss,speed_ms,0,0.001)
    |   movel(p[0.479375, -0.121887, -0.000100, 0.000000, -3.141593, 0.000000],accel_mss,speed_ms,0,0.001)
    |   movel(p[0.482068, -0.121876, -0.000100, 0.000000, -3.141593, 0.000000],accel_mss,speed_ms,0,blend_radius_m)
    |   movel(p[0.482985, -0.121906, -0.000100, 0.000000, -3.141593, 0.000000],accel_mss,speed_ms,0,0.000)
    |   movel(p[0.483437, -0.121986, -0.000100, 0.000000, -3.141593, 0.000000],accel_mss,speed_ms,0,0.000)
    |   movel(p[0.483622, -0.122168, -0.000100, 0.000000, -3.141593, 0.000000],accel_mss,speed_ms,0,0.000)
    |   movel(p[0.483699, -0.122335, -0.000100, 0.000000, -3.141593, 0.000000],accel_mss,speed_ms,0,0.000)
    |   movel(p[0.483891, -0.122630, -0.000100, 0.000000, -3.141593, 0.000000],accel_mss,speed_ms,0,0.000)
    |   movel(p[0.484132, -0.122967, -0.000100, 0.000000, -3.141593, 0.000000],accel_mss,speed_ms,0,0.000)
    |   movel(p[0.484399, -0.123309, -0.000100, 0.000000, -3.141593, 0.000000],accel_mss,speed_ms,0,0.000)
    |   movel(p[0.484739, -0.123726, -0.000100, 0.000000, -3.141593, 0.000000],accel_mss,speed_ms,0,0.000)
    |   movel(p[0.485079, -0.124143, -0.000100, 0.000000, -3.141593, 0.000000],accel_mss,speed_ms,0,0.000)
    |   movel(p[0.482428, -0.124121, -0.000100, 0.000000, -3.141593, 0.000000],accel_mss,speed_ms,0,blend_radius_m)
    |   movel(p[0.479777, -0.124099, -0.000100, 0.000000, -3.141593, 0.000000],accel_mss,speed_ms,0,blend_radius_m)
    |   movel(p[0.476315, -0.124063, -0.000100, 0.000000, -3.141593, 0.000000],accel_mss,speed_ms,0,blend_radius_m)
    |   movel(p[0.475075, -0.124014, -0.000100, 0.000000, -3.141593, 0.000000],accel_mss,speed_ms,0,0.000)
    |   movel(p[0.474369, -0.123910, -0.000100, 0.000000, -3.141593, 0.000000],accel_mss,speed_ms,0,0.000)
    |   movel(p[0.473801, -0.123700, -0.000100, 0.000000, -3.141593, 0.000000],accel_mss,speed_ms,0,0.000)
    |   movel(p[0.472940, -0.123141, -0.000100, 0.000000, -3.141593, 0.000000],accel_mss,speed_ms,0,0.000)
    |   movel(p[0.472253, -0.122457, -0.000100, 0.000000, -3.141593, 0.000000],accel_mss,speed_ms,0,0.000)
    |   movel(p[0.471743, -0.121649, -0.000100, 0.000000, -3.141593, 0.000000],accel_mss,speed_ms,0,0.000)
    |   movel(p[0.471406, -0.120719, -0.000100, 0.000000, -3.141593, 0.000000],accel_mss,speed_ms,0,0.000)
    |   movel(p[0.471305, -0.119638, -0.000100, 0.000000, -3.141593, 0.000000],accel_mss,speed_ms,0,0.000)
    |   movel(p[0.471520, -0.118504, -0.000100, 0.000000, -3.141593, 0.000000],accel_mss,speed_ms,0,0.000)
    |   movel(p[0.472020, -0.117441, -0.000100, 0.000000, -3.141593, 0.000000],accel_mss,speed_ms,0,0.000)
    |   speed_ms    = 0.050
    |   movel(p[0.472020, -0.117441, 0.003000, 0.000000, -3.141593, 0.000000],accel_mss,speed_ms,0,blend_radius_m)
    |   speed_ms    = 1.000
    |   movel(p[0.472020, -0.117441, 0.015000, 0.000000, -3.141593, 0.000000],accel_mss,speed_ms,0,blend_radius_m)
    | 
    |   movel(p[0.494039, -0.123170, 0.015000, 0.000000, -3.141593, 0.000000],accel_mss,speed_ms,0,blend_radius_m)
    | 
    |   movel(p[0.494039, -0.123170, 0.003000, 0.000000, -3.141593, 0.000000],accel_mss,speed_ms,0,blend_radius_m)
    |   speed_ms    = 0.050
    |   movel(p[0.494039, -0.123170, -0.000100, 0.000000, -3.141593, 0.000000],accel_mss,speed_ms,0,blend_radius_m)
    |   speed_ms    = 0.083
    |   movel(p[0.494303, -0.122907, -0.000100, 0.000000, -3.141593, 0.000000],accel_mss,speed_ms,0,0.000)
    |   movel(p[0.494566, -0.122644, -0.000100, 0.000000, -3.141593, 0.000000],accel_mss,speed_ms,0,0.000)
    |   movel(p[0.494829, -0.122380, -0.000100, 0.000000, -3.141593, 0.000000],accel_mss,speed_ms,0,0.000)
    |   movel(p[0.495092, -0.122117, -0.000100, 0.000000, -3.141593, 0.000000],accel_mss,speed_ms,0,0.000)
    |   movel(p[0.496201, -0.123208, -0.000100, 0.000000, -3.141593, 0.000000],accel_mss,speed_ms,0,0.001)
    |   movel(p[0.497309, -0.124299, -0.000100, 0.000000, -3.141593, 0.000000],accel_mss,speed_ms,0,0.001)
    |   movel(p[0.498271, -0.125226, -0.000100, 0.000000, -3.141593, 0.000000],accel_mss,speed_ms,0,0.001)
    |   movel(p[0.499053, -0.125933, -0.000100, 0.000000, -3.141593, 0.000000],accel_mss,speed_ms,0,0.000)
    |   movel(p[0.499672, -0.126448, -0.000100, 0.000000, -3.141593, 0.000000],accel_mss,speed_ms,0,0.000)
    |   movel(p[0.499953, -0.126587, -0.000100, 0.000000, -3.141593, 0.000000],accel_mss,speed_ms,0,0.000)
    |   movel(p[0.500833, -0.126543, -0.000100, 0.000000, -3.141593, 0.000000],accel_mss,speed_ms,0,0.000)
    |   movel(p[0.501661, -0.126023, -0.000100, 0.000000, -3.141593, 0.000000],accel_mss,speed_ms,0,0.000)
    |   movel(p[0.502188, -0.125207, -0.000100, 0.000000, -3.141593, 0.000000],accel_mss,speed_ms,0,0.000)
    |   movel(p[0.502235, -0.124338, -0.000100, 0.000000, -3.141593, 0.000000],accel_mss,speed_ms,0,0.000)
    |   movel(p[0.502111, -0.124095, -0.000100, 0.000000, -3.141593, 0.000000],accel_mss,speed_ms,0,0.000)
    |   movel(p[0.501530, -0.123413, -0.000100, 0.000000, -3.141593, 0.000000],accel_mss,speed_ms,0,0.000)
    |   movel(p[0.500801, -0.122606, -0.000100, 0.000000, -3.141593, 0.000000],accel_mss,speed_ms,0,0.000)
    |   movel(p[0.499940, -0.121707, -0.000100, 0.000000, -3.141593, 0.000000],accel_mss,speed_ms,0,0.000)
    |   movel(p[0.498841, -0.120587, -0.000100, 0.000000, -3.141593, 0.000000],accel_mss,speed_ms,0,0.001)
    |   movel(p[0.497742, -0.119467, -0.000100, 0.000000, -3.141593, 0.000000],accel_mss,speed_ms,0,0.001)
    |   movel(p[0.498006, -0.119204, -0.000100, 0.000000, -3.141593, 0.000000],accel_mss,speed_ms,0,0.000)
    |   movel(p[0.498269, -0.118941, -0.000100, 0.000000, -3.141593, 0.000000],accel_mss,speed_ms,0,0.000)
    |   movel(p[0.498532, -0.118678, -0.000100, 0.000000, -3.141593, 0.000000],accel_mss,speed_ms,0,0.000)
    |   movel(p[0.498795, -0.118414, -0.000100, 0.000000, -3.141593, 0.000000],accel_mss,speed_ms,0,0.000)
    |   movel(p[0.499917, -0.119562, -0.000100, 0.000000, -3.141593, 0.000000],accel_mss,speed_ms,0,0.001)
    |   movel(p[0.501038, -0.120710, -0.000100, 0.000000, -3.141593, 0.000000],accel_mss,speed_ms,0,0.001)
    |   movel(p[0.501916, -0.121629, -0.000100, 0.000000, -3.141593, 0.000000],accel_mss,speed_ms,0,0.001)
    |   movel(p[0.502699, -0.122491, -0.000100, 0.000000, -3.141593, 0.000000],accel_mss,speed_ms,0,0.000)
    |   movel(p[0.503333, -0.123229, -0.000100, 0.000000, -3.141593, 0.000000],accel_mss,speed_ms,0,0.000)
    |   movel(p[0.503541, -0.123552, -0.000100, 0.000000, -3.141593, 0.000000],accel_mss,speed_ms,0,0.000)
    |   movel(p[0.503769, -0.124410, -0.000100, 0.000000, -3.141593, 0.000000],accel_mss,speed_ms,0,0.000)
    |   movel(p[0.503669, -0.125281, -0.000100, 0.000000, -3.141593, 0.000000],accel_mss,speed_ms,0,0.000)
    |   movel(p[0.503225, -0.126161, -0.000100, 0.000000, -3.141593, 0.000000],accel_mss,speed_ms,0,0.000)
    |   movel(p[0.502441, -0.127048, -0.000100, 0.000000, -3.141593, 0.000000],accel_mss,speed_ms,0,0.000)
    |   movel(p[0.501588, -0.127725, -0.000100, 0.000000, -3.141593, 0.000000],accel_mss,speed_ms,0,0.000)
    |   movel(p[0.500799, -0.128089, -0.000100, 0.000000, -3.141593, 0.000000],accel_mss,speed_ms,0,0.000)
    |   movel(p[0.500024, -0.128161, -0.000100, 0.000000, -3.141593, 0.000000],accel_mss,speed_ms,0,0.000)
    |   movel(p[0.499218, -0.127960, -0.000100, 0.000000, -3.141593, 0.000000],accel_mss,speed_ms,0,0.000)
    |   movel(p[0.498905, -0.127770, -0.000100, 0.000000, -3.141593, 0.000000],accel_mss,speed_ms,0,0.000)
    |   movel(p[0.498167, -0.127137, -0.000100, 0.000000, -3.141593, 0.000000],accel_mss,speed_ms,0,0.000)
    |   movel(p[0.497301, -0.126351, -0.000100, 0.000000, -3.141593, 0.000000],accel_mss,speed_ms,0,0.000)
    |   movel(p[0.496367, -0.125456, -0.000100, 0.000000, -3.141593, 0.000000],accel_mss,speed_ms,0,0.001)
    |   movel(p[0.495203, -0.124313, -0.000100, 0.000000, -3.141593, 0.000000],accel_mss,speed_ms,0,0.001)
    |   movel(p[0.494039, -0.123170, -0.000100, 0.000000, -3.141593, 0.000000],accel_mss,speed_ms,0,0.001)
    |   speed_ms    = 0.050
    |   movel(p[0.494039, -0.123170, 0.003000, 0.000000, -3.141593, 0.000000],accel_mss,speed_ms,0,blend_radius_m)
    |   speed_ms    = 1.000
    |   movel(p[0.494039, -0.123170, 0.015000, 0.000000, -3.141593, 0.000000],accel_mss,speed_ms,0,blend_radius_m)
    | 
    |   movel(p[0.492326, -0.121867, 0.015000, 0.000000, -3.141593, 0.000000],accel_mss,speed_ms,0,0.001)
    | 
    |   movel(p[0.492326, -0.121867, 0.003000, 0.000000, -3.141593, 0.000000],accel_mss,speed_ms,0,blend_radius_m)
    |   speed_ms    = 0.050
    |   movel(p[0.492326, -0.121867, -0.000100, 0.000000, -3.141593, 0.000000],accel_mss,speed_ms,0,blend_radius_m)
    |   speed_ms    = 0.083
    |   movel(p[0.490992, -0.123320, -0.000100, 0.000000, -3.141593, 0.000000],accel_mss,speed_ms,0,0.001)
    |   movel(p[0.489114, -0.124039, -0.000100, 0.000000, -3.141593, 0.000000],accel_mss,speed_ms,0,0.001)
    |   movel(p[0.487111, -0.123872, -0.000100, 0.000000, -3.141593, 0.000000],accel_mss,speed_ms,0,0.001)
    |   movel(p[0.485431, -0.122849, -0.000100, 0.000000, -3.141593, 0.000000],accel_mss,speed_ms,0,0.001)
    |   movel(p[0.484869, -0.122164, -0.000100, 0.000000, -3.141593, 0.000000],accel_mss,speed_ms,0,0.000)
    |   movel(p[0.484495, -0.121423, -0.000100, 0.000000, -3.141593, 0.000000],accel_mss,speed_ms,0,0.000)
    |   movel(p[0.484267, -0.120521, -0.000100, 0.000000, -3.141593, 0.000000],accel_mss,speed_ms,0,0.000)
    |   movel(p[0.484151, -0.119329, -0.000100, 0.000000, -3.141593, 0.000000],accel_mss,speed_ms,0,0.000)
    |   movel(p[0.484114, -0.118541, -0.000100, 0.000000, -3.141593, 0.000000],accel_mss,speed_ms,0,0.000)
    |   movel(p[0.484076, -0.117754, -0.000100, 0.000000, -3.141593, 0.000000],accel_mss,speed_ms,0,0.000)
    |   movel(p[0.483344, -0.117732, -0.000100, 0.000000, -3.141593, 0.000000],accel_mss,speed_ms,0,0.000)
    |   movel(p[0.482613, -0.117711, -0.000100, 0.000000, -3.141593, 0.000000],accel_mss,speed_ms,0,0.000)
    |   movel(p[0.481882, -0.117690, -0.000100, 0.000000, -3.141593, 0.000000],accel_mss,speed_ms,0,0.000)
    |   movel(p[0.481151, -0.117668, -0.000100, 0.000000, -3.141593, 0.000000],accel_mss,speed_ms,0,0.000)
    |   movel(p[0.481151, -0.117108, -0.000100, 0.000000, -3.141593, 0.000000],accel_mss,speed_ms,0,0.000)
    |   movel(p[0.481151, -0.116548, -0.000100, 0.000000, -3.141593, 0.000000],accel_mss,speed_ms,0,0.000)
    |   movel(p[0.481151, -0.115989, -0.000100, 0.000000, -3.141593, 0.000000],accel_mss,speed_ms,0,0.000)
    |   movel(p[0.481151, -0.115429, -0.000100, 0.000000, -3.141593, 0.000000],accel_mss,speed_ms,0,0.000)
    |   movel(p[0.483216, -0.115429, -0.000100, 0.000000, -3.141593, 0.000000],accel_mss,speed_ms,0,0.001)
    |   movel(p[0.485282, -0.115429, -0.000100, 0.000000, -3.141593, 0.000000],accel_mss,speed_ms,0,0.001)
    |   movel(p[0.487348, -0.115429, -0.000100, 0.000000, -3.141593, 0.000000],accel_mss,speed_ms,0,0.001)
    |   movel(p[0.489414, -0.115429, -0.000100, 0.000000, -3.141593, 0.000000],accel_mss,speed_ms,0,0.001)
    |   movel(p[0.489392, -0.115973, -0.000100, 0.000000, -3.141593, 0.000000],accel_mss,speed_ms,0,0.000)
    |   movel(p[0.489370, -0.116516, -0.000100, 0.000000, -3.141593, 0.000000],accel_mss,speed_ms,0,0.000)
    |   movel(p[0.489348, -0.117060, -0.000100, 0.000000, -3.141593, 0.000000],accel_mss,speed_ms,0,0.000)
    |   movel(p[0.489326, -0.117604, -0.000100, 0.000000, -3.141593, 0.000000],accel_mss,speed_ms,0,0.000)
    |   movel(p[0.488587, -0.117625, -0.000100, 0.000000, -3.141593, 0.000000],accel_mss,speed_ms,0,0.000)
    |   movel(p[0.487849, -0.117647, -0.000100, 0.000000, -3.141593, 0.000000],accel_mss,speed_ms,0,0.000)
    |   movel(p[0.487111, -0.117669, -0.000100, 0.000000, -3.141593, 0.000000],accel_mss,speed_ms,0,0.000)
    |   movel(p[0.486373, -0.117690, -0.000100, 0.000000, -3.141593, 0.000000],accel_mss,speed_ms,0,0.000)
    |   movel(p[0.486399, -0.118431, -0.000100, 0.000000, -3.141593, 0.000000],accel_mss,speed_ms,0,0.000)
    |   movel(p[0.486424, -0.119173, -0.000100, 0.000000, -3.141593, 0.000000],accel_mss,speed_ms,0,0.000)
    |   movel(p[0.486466, -0.120042, -0.000100, 0.000000, -3.141593, 0.000000],accel_mss,speed_ms,0,0.000)
    |   movel(p[0.486528, -0.120480, -0.000100, 0.000000, -3.141593, 0.000000],accel_mss,speed_ms,0,0.000)
    |   movel(p[0.486644, -0.120777, -0.000100, 0.000000, -3.141593, 0.000000],accel_mss,speed_ms,0,0.000)
    |   movel(p[0.486851, -0.121056, -0.000100, 0.000000, -3.141593, 0.000000],accel_mss,speed_ms,0,0.000)
    |   movel(p[0.487734, -0.121682, -0.000100, 0.000000, -3.141593, 0.000000],accel_mss,speed_ms,0,0.000)
    |   movel(p[0.488735, -0.121857, -0.000100, 0.000000, -3.141593, 0.000000],accel_mss,speed_ms,0,0.000)
    |   movel(p[0.489671, -0.121545, -0.000100, 0.000000, -3.141593, 0.000000],accel_mss,speed_ms,0,0.000)
    |   movel(p[0.490376, -0.120812, -0.000100, 0.000000, -3.141593, 0.000000],accel_mss,speed_ms,0,0.000)
    |   movel(p[0.490547, -0.120370, -0.000100, 0.000000, -3.141593, 0.000000],accel_mss,speed_ms,0,0.000)
    |   movel(p[0.490637, -0.119732, -0.000100, 0.000000, -3.141593, 0.000000],accel_mss,speed_ms,0,0.000)
    |   movel(p[0.490686, -0.118629, -0.000100, 0.000000, -3.141593, 0.000000],accel_mss,speed_ms,0,0.000)
    |   movel(p[0.490722, -0.116059, -0.000100, 0.000000, -3.141593, 0.000000],accel_mss,speed_ms,0,blend_radius_m)
    |   movel(p[0.490758, -0.113259, -0.000100, 0.000000, -3.141593, 0.000000],accel_mss,speed_ms,0,blend_radius_m)
    |   movel(p[0.490804, -0.112342, -0.000100, 0.000000, -3.141593, 0.000000],accel_mss,speed_ms,0,0.000)
    |   movel(p[0.490899, -0.111894, -0.000100, 0.000000, -3.141593, 0.000000],accel_mss,speed_ms,0,0.000)
    |   movel(p[0.491097, -0.111689, -0.000100, 0.000000, -3.141593, 0.000000],accel_mss,speed_ms,0,0.000)
    |   movel(p[0.491268, -0.111600, -0.000100, 0.000000, -3.141593, 0.000000],accel_mss,speed_ms,0,0.000)
    |   movel(p[0.491540, -0.111413, -0.000100, 0.000000, -3.141593, 0.000000],accel_mss,speed_ms,0,0.000)
    |   movel(p[0.491846, -0.111179, -0.000100, 0.000000, -3.141593, 0.000000],accel_mss,speed_ms,0,0.000)
    |   movel(p[0.492145, -0.110926, -0.000100, 0.000000, -3.141593, 0.000000],accel_mss,speed_ms,0,0.000)
    |   movel(p[0.492505, -0.110609, -0.000100, 0.000000, -3.141593, 0.000000],accel_mss,speed_ms,0,0.000)
    |   movel(p[0.492865, -0.110291, -0.000100, 0.000000, -3.141593, 0.000000],accel_mss,speed_ms,0,0.000)
    |   movel(p[0.492843, -0.112982, -0.000100, 0.000000, -3.141593, 0.000000],accel_mss,speed_ms,0,blend_radius_m)
    |   movel(p[0.492820, -0.115672, -0.000100, 0.000000, -3.141593, 0.000000],accel_mss,speed_ms,0,blend_radius_m)
    |   movel(p[0.492798, -0.118363, -0.000100, 0.000000, -3.141593, 0.000000],accel_mss,speed_ms,0,blend_radius_m)
    |   movel(p[0.492776, -0.121054, -0.000100, 0.000000, -3.141593, 0.000000],accel_mss,speed_ms,0,blend_radius_m)
    |   movel(p[0.492551, -0.121460, -0.000100, 0.000000, -3.141593, 0.000000],accel_mss,speed_ms,0,0.000)
    |   movel(p[0.492326, -0.121867, -0.000100, 0.000000, -3.141593, 0.000000],accel_mss,speed_ms,0,0.000)
    |   speed_ms    = 0.050
    |   movel(p[0.492326, -0.121867, 0.003000, 0.000000, -3.141593, 0.000000],accel_mss,speed_ms,0,blend_radius_m)
    |   speed_ms    = 1.000
    |   movel(p[0.492326, -0.121867, 0.015000, 0.000000, -3.141593, 0.000000],accel_mss,speed_ms,0,blend_radius_m)
    | 
    |   movel(p[0.502602, -0.114608, 0.015000, 0.000000, -3.141593, 0.000000],accel_mss,speed_ms,0,blend_radius_m)
    | 
    |   movel(p[0.502602, -0.114608, 0.003000, 0.000000, -3.141593, 0.000000],accel_mss,speed_ms,0,blend_radius_m)
    |   speed_ms    = 0.050
    |   movel(p[0.502602, -0.114608, -0.000100, 0.000000, -3.141593, 0.000000],accel_mss,speed_ms,0,blend_radius_m)
    |   speed_ms    = 0.083
    |   movel(p[0.502864, -0.114345, -0.000100, 0.000000, -3.141593, 0.000000],accel_mss,speed_ms,0,0.000)
    |   movel(p[0.503127, -0.114082, -0.000100, 0.000000, -3.141593, 0.000000],accel_mss,speed_ms,0,0.000)
    |   movel(p[0.503390, -0.113820, -0.000100, 0.000000, -3.141593, 0.000000],accel_mss,speed_ms,0,0.000)
    |   movel(p[0.503653, -0.113557, -0.000100, 0.000000, -3.141593, 0.000000],accel_mss,speed_ms,0,0.000)
    |   movel(p[0.505158, -0.115062, -0.000100, 0.000000, -3.141593, 0.000000],accel_mss,speed_ms,0,0.001)
    |   movel(p[0.506663, -0.116568, -0.000100, 0.000000, -3.141593, 0.000000],accel_mss,speed_ms,0,0.001)
    |   movel(p[0.508169, -0.118073, -0.000100, 0.000000, -3.141593, 0.000000],accel_mss,speed_ms,0,0.001)
    |   movel(p[0.509674, -0.119578, -0.000100, 0.000000, -3.141593, 0.000000],accel_mss,speed_ms,0,0.001)
    |   movel(p[0.509474, -0.119816, -0.000100, 0.000000, -3.141593, 0.000000],accel_mss,speed_ms,0,0.000)
    |   movel(p[0.509274, -0.120054, -0.000100, 0.000000, -3.141593, 0.000000],accel_mss,speed_ms,0,0.000)
    |   movel(p[0.509108, -0.120236, -0.000100, 0.000000, -3.141593, 0.000000],accel_mss,speed_ms,0,0.000)
    |   movel(p[0.508941, -0.120389, -0.000100, 0.000000, -3.141593, 0.000000],accel_mss,speed_ms,0,0.000)
    |   movel(p[0.508792, -0.120501, -0.000100, 0.000000, -3.141593, 0.000000],accel_mss,speed_ms,0,0.000)
    |   movel(p[0.508585, -0.120483, -0.000100, 0.000000, -3.141593, 0.000000],accel_mss,speed_ms,0,0.000)
    |   movel(p[0.507709, -0.119659, -0.000100, 0.000000, -3.141593, 0.000000],accel_mss,speed_ms,0,0.000)
    |   movel(p[0.506713, -0.118703, -0.000100, 0.000000, -3.141593, 0.000000],accel_mss,speed_ms,0,0.001)
    |   movel(p[0.505565, -0.117568, -0.000100, 0.000000, -3.141593, 0.000000],accel_mss,speed_ms,0,0.001)
    |   movel(p[0.504083, -0.116088, -0.000100, 0.000000, -3.141593, 0.000000],accel_mss,speed_ms,0,0.001)
    |   movel(p[0.502602, -0.114608, -0.000100, 0.000000, -3.141593, 0.000000],accel_mss,speed_ms,0,0.001)
    |   speed_ms    = 0.050
    |   movel(p[0.502602, -0.114608, 0.003000, 0.000000, -3.141593, 0.000000],accel_mss,speed_ms,0,blend_radius_m)
    |   speed_ms    = 1.000
    |   movel(p[0.502602, -0.114608, 0.015000, 0.000000, -3.141593, 0.000000],accel_mss,speed_ms,0,blend_radius_m)
    | 
    |   movel(p[0.506318, -0.113033, 0.015000, 0.000000, -3.141593, 0.000000],accel_mss,speed_ms,0,blend_radius_m)
    | 
    |   movel(p[0.506318, -0.113033, 0.003000, 0.000000, -3.141593, 0.000000],accel_mss,speed_ms,0,blend_radius_m)
    |   speed_ms    = 0.050
    |   movel(p[0.506318, -0.113033, -0.000100, 0.000000, -3.141593, 0.000000],accel_mss,speed_ms,0,blend_radius_m)
    |   speed_ms    = 0.083
    |   movel(p[0.506196, -0.112240, -0.000100, 0.000000, -3.141593, 0.000000],accel_mss,speed_ms,0,0.000)
    |   movel(p[0.506287, -0.111464, -0.000100, 0.000000, -3.141593, 0.000000],accel_mss,speed_ms,0,0.000)
    |   movel(p[0.506588, -0.110660, -0.000100, 0.000000, -3.141593, 0.000000],accel_mss,speed_ms,0,0.000)
    |   movel(p[0.507392, -0.109520, -0.000100, 0.000000, -3.141593, 0.000000],accel_mss,speed_ms,0,0.001)
    |   movel(p[0.508467, -0.108736, -0.000100, 0.000000, -3.141593, 0.000000],accel_mss,speed_ms,0,0.001)
    |   movel(p[0.509654, -0.108414, -0.000100, 0.000000, -3.141593, 0.000000],accel_mss,speed_ms,0,0.000)
    |   movel(p[0.510787, -0.108599, -0.000100, 0.000000, -3.141593, 0.000000],accel_mss,speed_ms,0,0.000)
    |   movel(p[0.511124, -0.108751, -0.000100, 0.000000, -3.141593, 0.000000],accel_mss,speed_ms,0,0.000)
    |   movel(p[0.511218, -0.108847, -0.000100, 0.000000, -3.141593, 0.000000],accel_mss,speed_ms,0,0.000)
    |   movel(p[0.511219, -0.108975, -0.000100, 0.000000, -3.141593, 0.000000],accel_mss,speed_ms,0,0.000)
    |   movel(p[0.511083, -0.109264, -0.000100, 0.000000, -3.141593, 0.000000],accel_mss,speed_ms,0,0.000)
    |   movel(p[0.510856, -0.109630, -0.000100, 0.000000, -3.141593, 0.000000],accel_mss,speed_ms,0,0.000)
    |   movel(p[0.510631, -0.109820, -0.000100, 0.000000, -3.141593, 0.000000],accel_mss,speed_ms,0,0.000)
    |   movel(p[0.510314, -0.109911, -0.000100, 0.000000, -3.141593, 0.000000],accel_mss,speed_ms,0,0.000)
    |   movel(p[0.509736, -0.109945, -0.000100, 0.000000, -3.141593, 0.000000],accel_mss,speed_ms,0,0.000)
    |   movel(p[0.509395, -0.109969, -0.000100, 0.000000, -3.141593, 0.000000],accel_mss,speed_ms,0,0.000)
    |   movel(p[0.509071, -0.110028, -0.000100, 0.000000, -3.141593, 0.000000],accel_mss,speed_ms,0,0.000)
    |   movel(p[0.508788, -0.110117, -0.000100, 0.000000, -3.141593, 0.000000],accel_mss,speed_ms,0,0.000)
    |   movel(p[0.508570, -0.110231, -0.000100, 0.000000, -3.141593, 0.000000],accel_mss,speed_ms,0,0.000)
    |   movel(p[0.508168, -0.110618, -0.000100, 0.000000, -3.141593, 0.000000],accel_mss,speed_ms,0,0.000)
    |   movel(p[0.507830, -0.111196, -0.000100, 0.000000, -3.141593, 0.000000],accel_mss,speed_ms,0,0.000)
    |   movel(p[0.507622, -0.111818, -0.000100, 0.000000, -3.141593, 0.000000],accel_mss,speed_ms,0,0.000)
    |   movel(p[0.507613, -0.112337, -0.000100, 0.000000, -3.141593, 0.000000],accel_mss,speed_ms,0,0.000)
    |   movel(p[0.507824, -0.112949, -0.000100, 0.000000, -3.141593, 0.000000],accel_mss,speed_ms,0,0.000)
    |   movel(p[0.508250, -0.113628, -0.000100, 0.000000, -3.141593, 0.000000],accel_mss,speed_ms,0,0.000)
    |   movel(p[0.508819, -0.114285, -0.000100, 0.000000, -3.141593, 0.000000],accel_mss,speed_ms,0,0.000)
    |   movel(p[0.509467, -0.114832, -0.000100, 0.000000, -3.141593, 0.000000],accel_mss,speed_ms,0,0.000)
    |   movel(p[0.509928, -0.115141, -0.000100, 0.000000, -3.141593, 0.000000],accel_mss,speed_ms,0,0.000)
    |   movel(p[0.510271, -0.115314, -0.000100, 0.000000, -3.141593, 0.000000],accel_mss,speed_ms,0,0.000)
    |   movel(p[0.510597, -0.115400, -0.000100, 0.000000, -3.141593, 0.000000],accel_mss,speed_ms,0,0.000)
    |   movel(p[0.510988, -0.115428, -0.000100, 0.000000, -3.141593, 0.000000],accel_mss,speed_ms,0,0.000)
    |   movel(p[0.511871, -0.115265, -0.000100, 0.000000, -3.141593, 0.000000],accel_mss,speed_ms,0,0.000)
    |   movel(p[0.512570, -0.114801, -0.000100, 0.000000, -3.141593, 0.000000],accel_mss,speed_ms,0,0.000)
    |   movel(p[0.512984, -0.114101, -0.000100, 0.000000, -3.141593, 0.000000],accel_mss,speed_ms,0,0.000)
    |   movel(p[0.513059, -0.113267, -0.000100, 0.000000, -3.141593, 0.000000],accel_mss,speed_ms,0,0.000)
    |   movel(p[0.513023, -0.113015, -0.000100, 0.000000, -3.141593, 0.000000],accel_mss,speed_ms,0,0.000)
    |   movel(p[0.512978, -0.112766, -0.000100, 0.000000, -3.141593, 0.000000],accel_mss,speed_ms,0,0.000)
    |   movel(p[0.512930, -0.112550, -0.000100, 0.000000, -3.141593, 0.000000],accel_mss,speed_ms,0,0.000)
    |   movel(p[0.512888, -0.112421, -0.000100, 0.000000, -3.141593, 0.000000],accel_mss,speed_ms,0,0.000)
    |   movel(p[0.512878, -0.112300, -0.000100, 0.000000, -3.141593, 0.000000],accel_mss,speed_ms,0,0.000)
    |   movel(p[0.512939, -0.112184, -0.000100, 0.000000, -3.141593, 0.000000],accel_mss,speed_ms,0,0.000)
    |   movel(p[0.513083, -0.112065, -0.000100, 0.000000, -3.141593, 0.000000],accel_mss,speed_ms,0,0.000)
    |   movel(p[0.513326, -0.111934, -0.000100, 0.000000, -3.141593, 0.000000],accel_mss,speed_ms,0,0.000)
    |   movel(p[0.513826, -0.111724, -0.000100, 0.000000, -3.141593, 0.000000],accel_mss,speed_ms,0,0.000)
